LIN {X 0,Y 453.11,Z 853.7,A -85,B 0,C 180,E1 14752.247,E2 14752.247} C_VEL
LIN {X 0,Y 449.682,Z 846.893,A -85,B 0,C 180,E1 14758.978,E2 14758.978} C_VEL
LIN {X 0,Y 456.132,Z 857.359,A -85,B 0,C 180,E1 14770.845,E2 14770.845} C_VEL
LIN {X 0,Y 467.562,Z 871.986,A -85,B 0,C 180,E1 14777.472,E2 14777.472} C_VEL
LIN {X 0,Y 488.075,Z 901.104,A -85,B 0,C 180,E1 14785.371,E2 14785.371} C_VEL
LIN {X 0,Y 511.745,Z 944.514,A -85,B 0,C 180,E1 14792.88,E2 14792.88} C_VEL
LIN {X 0,Y 522.504,Z 975.983,A -85,B 0,C 180,E1 14796.793,E2 14796.793} C_VEL
LIN {X 0,Y 504.777,Z 1049.312,A -85,B 0,C 180,E1 14800.922,E2 14800.922} C_VEL
LIN {X 0,Y 484.838,Z 1113.765,A -85,B 0,C 180,E1 14806.768,E2 14806.768} C_VEL
LIN {X 0,Y 466.012,Z 1168.211,A -85,B 0,C 180,E1 14814.348,E2 14814.348} C_VEL
LIN {X 0,Y 452.106,Z 1211.205,A -85,B 0,C 180,E1 14823.581,E2 14823.581} C_VEL
LIN {X 0,Y 445.258,Z 1240.185,A -85,B 0,C 180,E1 14833.662,E2 14833.662} C_VEL
LIN {X 0,Y 443.189,Z 1254.354,A -85,B 0,C 180,E1 14843.114,E2 14843.114} C_VEL
LIN {X 0,Y 443.168,Z 1257.3,A -85,B 0,C 180,E1 14850.981,E2 14850.981} C_VEL
LIN {X 0,Y 443.526,Z 1251.078,A -85,B 0,C 180,E1 14859.854,E2 14859.854} C_VEL
LIN {X 0,Y 446.199,Z 1232.875,A -85,B 0,C 180,E1 14869.373,E2 14869.373} C_VEL
LIN {X 0,Y 455.013,Z 1201.001,A -85,B 0,C 180,E1 14878.932,E2 14878.932} C_VEL
LIN {X 0,Y 470.637,Z 1154.491,A -85,B 0,C 180,E1 14887.802,E2 14887.802} C_VEL
LIN {X 0,Y 490.557,Z 1096.151,A -85,B 0,C 180,E1 14895.007,E2 14895.007} C_VEL
LIN {X 0,Y 510.312,Z 1029.556,A -85,B 0,C 180,E1 14900.284,E2 14900.284} C_VEL
LIN {X 0,Y 522.312,Z 970.799,A -85,B 0,C 180,E1 14903.513,E2 14903.513} C_VEL
LIN {X 0,Y 500.816,Z 922.884,A -85,B 0,C 180,E1 14910.405,E2 14910.405} C_VEL
LIN {X 0,Y 478.038,Z 886.237,A -85,B 0,C 180,E1 14918.038,E2 14918.038} C_VEL
LIN {X 0,Y 460.008,Z 861.655,A -85,B 0,C 180,E1 14926.343,E2 14926.343} C_VEL
LIN {X 0,Y 453.526,Z 853.849,A -85,B 0,C 180,E1 14931.155,E2 14931.155} C_VEL
LIN {X 0,Y 449.33,Z 846.815,A -85,B 0,C 180,E1 14939.088,E2 14939.088} C_VEL
LIN {X 0,Y 455.483,Z 855.768,A -85,B 0,C 180,E1 14950.006,E2 14950.006} C_VEL
LIN {X 0,Y 468.677,Z 873.827,A -85,B 0,C 180,E1 14957.65,E2 14957.65} C_VEL
LIN {X 0,Y 490.163,Z 903.109,A -85,B 0,C 180,E1 14965.368,E2 14965.368} C_VEL
LIN {X 0,Y 516.111,Z 949.406,A -85,B 0,C 180,E1 14972.898,E2 14972.898} C_VEL
LIN {X 0,Y 525.972,Z 974.905,A -85,B 0,C 180,E1 14975.93,E2 14975.93} C_VEL
LIN {X 0,Y 510.004,Z 1047.435,A -85,B 0,C 180,E1 14979.293,E2 14979.293} C_VEL
LIN {X 0,Y 490.013,Z 1116.733,A -85,B 0,C 180,E1 14984.599,E2 14984.599} C_VEL
LIN {X 0,Y 470.658,Z 1176.48,A -85,B 0,C 180,E1 14991.727,E2 14991.727} C_VEL
LIN {X 0,Y 455.499,Z 1224.574,A -85,B 0,C 180,E1 15000.429,E2 15000.429} C_VEL
LIN {X 0,Y 446.704,Z 1259.254,A -85,B 0,C 180,E1 15010.133,E2 15010.133} C_VEL
LIN {X 0,Y 443.508,Z 1278.435,A -85,B 0,C 180,E1 15019.149,E2 15019.149} C_VEL
LIN {X 0,Y 443.111,Z 1285.921,A -85,B 0,C 180,E1 15027.055,E2 15027.055} C_VEL
LIN {X 0,Y 443.189,Z 1284.856,A -85,B 0,C 180,E1 15034.913,E2 15034.913} C_VEL
LIN {X 0,Y 443.981,Z 1273.992,A -85,B 0,C 180,E1 15043.49,E2 15043.49} C_VEL
LIN {X 0,Y 437.709,Z 1265,A -85,B 0,C 180,E1 15047.886,E2 15047.886} C_VEL
LIN {X 0,Y 445.554,Z 1232.734,A -85,B 0,C 180,E1 15058.106,E2 15058.106} C_VEL
LIN {X 0,Y 460.411,Z 1186.788,A -85,B 0,C 180,E1 15067.293,E2 15067.293} C_VEL
LIN {X 0,Y 480.299,Z 1128.807,A -85,B 0,C 180,E1 15074.859,E2 15074.859} C_VEL
LIN {X 0,Y 501.097,Z 1060.927,A -85,B 0,C 180,E1 15080.584,E2 15080.584} C_VEL
LIN {X 0,Y 519.127,Z 985.374,A -85,B 0,C 180,E1 15084.445,E2 15084.445} C_VEL
LIN {X 0,Y 519.955,Z 974.55,A -85,B 0,C 180,E1 15085.007,E2 15085.007} C_VEL
LIN {X 0,Y 497.411,Z 926.333,A -85,B 0,C 180,E1 15091.89,E2 15091.89} C_VEL
LIN {X 0,Y 474.399,Z 890.834,A -85,B 0,C 180,E1 15099.591,E2 15099.591} C_VEL
LIN {X 0,Y 457.866,Z 869.113,A -85,B 0,C 180,E1 15107.615,E2 15107.615} C_VEL
LIN {X 0,Y 451.9,Z 861.515,A -85,B 0,C 180,E1 15112.469,E2 15112.469} C_VEL
LIN {X 0,Y 448.631,Z 854.888,A -85,B 0,C 180,E1 15120.913,E2 15120.913} C_VEL
LIN {X 0,Y 455.13,Z 865.662,A -85,B 0,C 180,E1 15130.869,E2 15130.869} C_VEL
LIN {X 0,Y 466.056,Z 880.022,A -85,B 0,C 180,E1 15137.347,E2 15137.347} C_VEL
LIN {X 0,Y 486.826,Z 910.227,A -85,B 0,C 180,E1 15145.543,E2 15145.543} C_VEL
LIN {X 0,Y 508.661,Z 953.325,A -85,B 0,C 180,E1 15152.921,E2 15152.921} C_VEL
LIN {X 0,Y 517.223,Z 978.635,A -85,B 0,C 180,E1 15156.18,E2 15156.18} C_VEL
LIN {X 0,Y 499.121,Z 1050.75,A -85,B 0,C 180,E1 15160.297,E2 15160.297} C_VEL
LIN {X 0,Y 478.45,Z 1115.183,A -85,B 0,C 180,E1 15166.219,E2 15166.219} C_VEL
LIN {X 0,Y 459.135,Z 1168.858,A -85,B 0,C 180,E1 15173.807,E2 15173.807} C_VEL
LIN {X 0,Y 444.616,Z 1211.478,A -85,B 0,C 180,E1 15183.101,E2 15183.101} C_VEL
LIN {X 0,Y 437.447,Z 1240.451,A -85,B 0,C 180,E1 15193.362,E2 15193.362} C_VEL
LIN {X 0,Y 435.219,Z 1254.617,A -85,B 0,C 180,E1 15202.987,E2 15202.987} C_VEL
LIN {X 0,Y 435.171,Z 1257.563,A -85,B 0,C 180,E1 15210.999,E2 15210.999} C_VEL
LIN {X 0,Y 435.567,Z 1251.344,A -85,B 0,C 180,E1 15220.036,E2 15220.036} C_VEL
LIN {X 0,Y 438.475,Z 1233.146,A -85,B 0,C 180,E1 15229.728,E2 15229.728} C_VEL
LIN {X 0,Y 447.767,Z 1201.276,A -85,B 0,C 180,E1 15239.446,E2 15239.446} C_VEL
LIN {X 0,Y 464.103,Z 1154.767,A -85,B 0,C 180,E1 15248.431,E2 15248.431} C_VEL
LIN {X 0,Y 484.889,Z 1096.018,A -85,B 0,C 180,E1 15255.738,E2 15255.738} C_VEL
LIN {X 0,Y 504.973,Z 1030.479,A -85,B 0,C 180,E1 15260.953,E2 15260.953} C_VEL
LIN {X 0,Y 516.768,Z 974.458,A -85,B 0,C 180,E1 15264.101,E2 15264.101} C_VEL
LIN {X 0,Y 496.134,Z 927.061,A -85,B 0,C 180,E1 15271.146,E2 15271.146} C_VEL
LIN {X 0,Y 473.874,Z 890.484,A -85,B 0,C 180,E1 15279.129,E2 15279.129} C_VEL
LIN {X 0,Y 457.673,Z 868.684,A -85,B 0,C 180,E1 15287.126,E2 15287.126} C_VEL
LIN {X 0,Y 452.049,Z 861.472,A -85,B 0,C 180,E1 15291.612,E2 15291.612} C_VEL
LIN {X 0,Y 448.355,Z 854.755,A -85,B 0,C 180,E1 15299.086,E2 15299.086} C_VEL
LIN {X 0,Y 454.259,Z 863.811,A -85,B 0,C 180,E1 15309.851,E2 15309.851} C_VEL
LIN {X 0,Y 467.341,Z 881.776,A -85,B 0,C 180,E1 15317.531,E2 15317.531} C_VEL
LIN {X 0,Y 488.148,Z 911.534,A -85,B 0,C 180,E1 15325.295,E2 15325.295} C_VEL
LIN {X 0,Y 512.404,Z 956.503,A -85,B 0,C 180,E1 15332.685,E2 15332.685} C_VEL
LIN {X 0,Y 520.374,Z 979.416,A -85,B 0,C 180,E1 15335.378,E2 15335.378} C_VEL
LIN {X 0,Y 503.728,Z 1051.271,A -85,B 0,C 180,E1 15338.825,E2 15338.825} C_VEL
LIN {X 0,Y 482.851,Z 1120.512,A -85,B 0,C 180,E1 15344.293,E2 15344.293} C_VEL
LIN {X 0,Y 463.009,Z 1179.262,A -85,B 0,C 180,E1 15351.541,E2 15351.541} C_VEL
LIN {X 0,Y 447.361,Z 1227.03,A -85,B 0,C 180,E1 15360.525,E2 15360.525} C_VEL
LIN {X 0,Y 438.59,Z 1260.356,A -85,B 0,C 180,E1 15370.277,E2 15370.277} C_VEL
LIN {X 0,Y 435.425,Z 1279.547,A -85,B 0,C 180,E1 15379.961,E2 15379.961} C_VEL
LIN {X 0,Y 435.469,Z 1286.143,A -85,B 0,C 180,E1 15389.002,E2 15389.002} C_VEL
LIN {X 0,Y 435.223,Z 1282.035,A -85,B 0,C 180,E1 15398.021,E2 15398.021} C_VEL
LIN {X 0,Y 437.709,Z 1265,A -85,B 0,C 180,E1 15407.886,E2 15407.886} C_VEL
LIN {X 0,Y 431.738,Z 1254.138,A -85,B 0,C 180,E1 15412.282,E2 15412.282} C_VEL
LIN {X 0,Y 442.101,Z 1219.334,A -85,B 0,C 180,E1 15421.759,E2 15421.759} C_VEL
LIN {X 0,Y 459.976,Z 1168.875,A -85,B 0,C 180,E1 15430.636,E2 15430.636} C_VEL
LIN {X 0,Y 481.519,Z 1107.411,A -85,B 0,C 180,E1 15437.644,E2 15437.644} C_VEL
LIN {X 0,Y 501.982,Z 1039.364,A -85,B 0,C 180,E1 15442.593,E2 15442.593} C_VEL
LIN {X 0,Y 514.55,Z 978.138,A -85,B 0,C 180,E1 15445.62,E2 15445.62} C_VEL
LIN {X 0,Y 493.082,Z 931.355,A -85,B 0,C 180,E1 15452.528,E2 15452.528} C_VEL
LIN {X 0,Y 471.954,Z 897.803,A -85,B 0,C 180,E1 15460.033,E2 15460.033} C_VEL
LIN {X 0,Y 456.328,Z 876.653,A -85,B 0,C 180,E1 15467.951,E2 15467.951} C_VEL
LIN {X 0,Y 450.479,Z 869.111,A -85,B 0,C 180,E1 15472.932,E2 15472.932} C_VEL
LIN {X 0,Y 447.656,Z 862.828,A -85,B 0,C 180,E1 15480.915,E2 15480.915} C_VEL
LIN {X 0,Y 453.995,Z 873.676,A -85,B 0,C 180,E1 15490.779,E2 15490.779} C_VEL
LIN {X 0,Y 464.875,Z 888.499,A -85,B 0,C 180,E1 15497.392,E2 15497.392} C_VEL
LIN {X 0,Y 484.206,Z 918.023,A -85,B 0,C 180,E1 15505.394,E2 15505.394} C_VEL
LIN {X 0,Y 504.697,Z 960.166,A -85,B 0,C 180,E1 15512.7,E2 15512.7} C_VEL
LIN {X 0,Y 511.792,Z 982.53,A -85,B 0,C 180,E1 15515.615,E2 15515.615} C_VEL
LIN {X 0,Y 492.699,Z 1054.947,A -85,B 0,C 180,E1 15519.854,E2 15519.854} C_VEL
LIN {X 0,Y 471.361,Z 1118.752,A -85,B 0,C 180,E1 15525.899,E2 15525.899} C_VEL
LIN {X 0,Y 450.971,Z 1173.22,A -85,B 0,C 180,E1 15533.906,E2 15533.906} C_VEL
LIN {X 0,Y 436.26,Z 1215.391,A -85,B 0,C 180,E1 15543.66,E2 15543.66} C_VEL
LIN {X 0,Y 429.385,Z 1241.838,A -85,B 0,C 180,E1 15553.569,E2 15553.569} C_VEL
LIN {X 0,Y 427.232,Z 1254.881,A -85,B 0,C 180,E1 15562.855,E2 15562.855} C_VEL
LIN {X 0,Y 427.202,Z 1257.824,A -85,B 0,C 180,E1 15571.017,E2 15571.017} C_VEL
LIN {X 0,Y 427.586,Z 1251.611,A -85,B 0,C 180,E1 15580.225,E2 15580.225} C_VEL
LIN {X 0,Y 430.757,Z 1233.435,A -85,B 0,C 180,E1 15590.089,E2 15590.089} C_VEL
LIN {X 0,Y 440.547,Z 1201.552,A -85,B 0,C 180,E1 15599.977,E2 15599.977} C_VEL
LIN {X 0,Y 457.389,Z 1155.709,A -85,B 0,C 180,E1 15608.972,E2 15608.972} C_VEL
LIN {X 0,Y 478.774,Z 1097.425,A -85,B 0,C 180,E1 15616.331,E2 15616.331} C_VEL
LIN {X 0,Y 499.892,Z 1030.798,A -85,B 0,C 180,E1 15621.672,E2 15621.672} C_VEL
LIN {X 0,Y 511.857,Z 979.714,A -85,B 0,C 180,E1 15624.486,E2 15624.486} C_VEL
LIN {X 0,Y 492.306,Z 932.966,A -85,B 0,C 180,E1 15631.591,E2 15631.591} C_VEL
LIN {X 0,Y 471.233,Z 897.38,A -85,B 0,C 180,E1 15639.561,E2 15639.561} C_VEL
LIN {X 0,Y 455.949,Z 876.053,A -85,B 0,C 180,E1 15647.565,E2 15647.565} C_VEL
LIN {X 0,Y 450.835,Z 869.282,A -85,B 0,C 180,E1 15651.833,E2 15651.833} C_VEL
LIN {X 0,Y 447.381,Z 862.695,A -85,B 0,C 180,E1 15659.084,E2 15659.084} C_VEL
LIN {X 0,Y 453.357,Z 872.65,A -85,B 0,C 180,E1 15669.992,E2 15669.992} C_VEL
LIN {X 0,Y 465.347,Z 889.013,A -85,B 0,C 180,E1 15677.181,E2 15677.181} C_VEL
LIN {X 0,Y 485.623,Z 918.952,A -85,B 0,C 180,E1 15685.063,E2 15685.063} C_VEL
LIN {X 0,Y 508.669,Z 963.487,A -85,B 0,C 180,E1 15692.456,E2 15692.456} C_VEL
LIN {X 0,Y 514.971,Z 982.994,A -85,B 0,C 180,E1 15694.776,E2 15694.776} C_VEL
LIN {X 0,Y 497.853,Z 1053.719,A -85,B 0,C 180,E1 15698.257,E2 15698.257} C_VEL
LIN {X 0,Y 476.308,Z 1122.453,A -85,B 0,C 180,E1 15703.794,E2 15703.794} C_VEL
LIN {X 0,Y 456.004,Z 1180.218,A -85,B 0,C 180,E1 15711.071,E2 15711.071} C_VEL
LIN {X 0,Y 439.71,Z 1227.863,A -85,B 0,C 180,E1 15720.245,E2 15720.245} C_VEL
LIN {X 0,Y 430.453,Z 1261.457,A -85,B 0,C 180,E1 15730.425,E2 15730.425} C_VEL
LIN {X 0,Y 427.443,Z 1279.281,A -85,B 0,C 180,E1 15739.772,E2 15739.772} C_VEL
LIN {X 0,Y 427.486,Z 1285.881,A -85,B 0,C 180,E1 15748.983,E2 15748.983} C_VEL
LIN {X 0,Y 427.261,Z 1281.771,A -85,B 0,C 180,E1 15758.171,E2 15758.171} C_VEL
LIN {X 0,Y 430.028,Z 1264.044,A -85,B 0,C 180,E1 15768.526,E2 15768.526} C_VEL
LIN {X 0,Y 431.738,Z 1254.138,A -85,B 0,C 180,E1 15772.282,E2 15772.282} C_VEL
LIN {X 0,Y 428.136,Z 1241.283,A -85,B 0,C 180,E1 15776.671,E2 15776.671} C_VEL
LIN {X 0,Y 442.508,Z 1198.865,A -85,B 0,C 180,E1 15786.394,E2 15786.394} C_VEL
LIN {X 0,Y 463.058,Z 1143.42,A -85,B 0,C 180,E1 15794.606,E2 15794.606} C_VEL
LIN {X 0,Y 485.732,Z 1077.138,A -85,B 0,C 180,E1 15800.89,E2 15800.89} C_VEL
LIN {X 0,Y 505.9,Z 1003.625,A -85,B 0,C 180,E1 15805.141,E2 15805.141} C_VEL
LIN {X 0,Y 509.324,Z 982.117,A -85,B 0,C 180,E1 15806.2,E2 15806.2} C_VEL
LIN {X 0,Y 488.656,Z 936.006,A -85,B 0,C 180,E1 15813.237,E2 15813.237} C_VEL
LIN {X 0,Y 468.949,Z 904.053,A -85,B 0,C 180,E1 15820.699,E2 15820.699} C_VEL
LIN {X 0,Y 454.583,Z 884.034,A -85,B 0,C 180,E1 15828.392,E2 15828.392} C_VEL
LIN {X 0,Y 449.084,Z 876.743,A -85,B 0,C 180,E1 15833.397,E2 15833.397} C_VEL
LIN {X 0,Y 446.683,Z 870.754,A -85,B 0,C 180,E1 15840.917,E2 15840.917} C_VEL
LIN {X 0,Y 452.859,Z 881.852,A -85,B 0,C 180,E1 15850.806,E2 15850.806} C_VEL
LIN {X 0,Y 465.789,Z 899.557,A -85,B 0,C 180,E1 15858.522,E2 15858.522} C_VEL
LIN {X 0,Y 485.836,Z 933.76,A -85,B 0,C 180,E1 15866.867,E2 15866.867} C_VEL
LIN {X 0,Y 504.507,Z 977.636,A -85,B 0,C 180,E1 15874.019,E2 15874.019} C_VEL
LIN {X 0,Y 505.912,Z 988.262,A -85,B 0,C 180,E1 15875.126,E2 15875.126} C_VEL
LIN {X 0,Y 485.863,Z 1060.395,A -85,B 0,C 180,E1 15879.521,E2 15879.521} C_VEL
LIN {X 0,Y 463.572,Z 1123.832,A -85,B 0,C 180,E1 15885.777,E2 15885.777} C_VEL
LIN {X 0,Y 443.176,Z 1176.189,A -85,B 0,C 180,E1 15893.798,E2 15893.798} C_VEL
LIN {X 0,Y 428.288,Z 1217.361,A -85,B 0,C 180,E1 15903.699,E2 15903.699} C_VEL
LIN {X 0,Y 420.937,Z 1244.017,A -85,B 0,C 180,E1 15914.306,E2 15914.306} C_VEL
LIN {X 0,Y 419.162,Z 1256.093,A -85,B 0,C 180,E1 15923.903,E2 15923.903} C_VEL
LIN {X 0,Y 419.202,Z 1257.635,A -85,B 0,C 180,E1 15933.113,E2 15933.113} C_VEL
LIN {X 0,Y 419.846,Z 1249.304,A -85,B 0,C 180,E1 15942.354,E2 15942.354} C_VEL
LIN {X 0,Y 424.922,Z 1228.23,A -85,B 0,C 180,E1 15952.585,E2 15952.585} C_VEL
LIN {X 0,Y 436.897,Z 1193.077,A -85,B 0,C 180,E1 15962.587,E2 15962.587} C_VEL
LIN {X 0,Y 455.094,Z 1145.757,A -85,B 0,C 180,E1 15971.193,E2 15971.193} C_VEL
LIN {X 0,Y 477.176,Z 1086.488,A -85,B 0,C 180,E1 15978.141,E2 15978.141} C_VEL
LIN {X 0,Y 498.343,Z 1018.96,A -85,B 0,C 180,E1 15983.144,E2 15983.144} C_VEL
LIN {X 0,Y 506.159,Z 982.556,A -85,B 0,C 180,E1 15985.203,E2 15985.203} C_VEL
LIN {X 0,Y 487.494,Z 937.272,A -85,B 0,C 180,E1 15992.359,E2 15992.359} C_VEL
LIN {X 0,Y 468.289,Z 903.91,A -85,B 0,C 180,E1 16000.107,E2 16000.107} C_VEL
LIN {X 0,Y 454.043,Z 883.251,A -85,B 0,C 180,E1 16008.063,E2 16008.063} C_VEL
LIN {X 0,Y 449.166,Z 876.737,A -85,B 0,C 180,E1 16012.535,E2 16012.535} C_VEL
LIN {X 0,Y 446.406,Z 870.635,A -85,B 0,C 180,E1 16019.082,E2 16019.082} C_VEL
LIN {X 0,Y 452.407,Z 881.126,A -85,B 0,C 180,E1 16030.075,E2 16030.075} C_VEL
LIN {X 0,Y 464.066,Z 897.184,A -85,B 0,C 180,E1 16037.168,E2 16037.168} C_VEL
LIN {X 0,Y 483.946,Z 927.901,A -85,B 0,C 180,E1 16045.164,E2 16045.164} C_VEL
LIN {X 0,Y 504.916,Z 970.827,A -85,B 0,C 180,E1 16052.291,E2 16052.291} C_VEL
LIN {X 0,Y 509.389,Z 987.554,A -85,B 0,C 180,E1 16054.207,E2 16054.207} C_VEL
LIN {X 0,Y 491.278,Z 1059.063,A -85,B 0,C 180,E1 16057.866,E2 16057.866} C_VEL
LIN {X 0,Y 469.06,Z 1126.651,A -85,B 0,C 180,E1 16063.514,E2 16063.514} C_VEL
LIN {X 0,Y 447.703,Z 1184.738,A -85,B 0,C 180,E1 16071.148,E2 16071.148} C_VEL
LIN {X 0,Y 431.377,Z 1230.805,A -85,B 0,C 180,E1 16080.483,E2 16080.483} C_VEL
LIN {X 0,Y 421.966,Z 1263.766,A -85,B 0,C 180,E1 16091.108,E2 16091.108} C_VEL
LIN {X 0,Y 419.361,Z 1280.267,A -85,B 0,C 180,E1 16100.625,E2 16100.625} C_VEL
LIN {X 0,Y 419.478,Z 1285.618,A -85,B 0,C 180,E1 16108.964,E2 16108.964} C_VEL
LIN {X 0,Y 419.289,Z 1281.506,A -85,B 0,C 180,E1 16118.328,E2 16118.328} C_VEL
LIN {X 0,Y 422.198,Z 1263.772,A -85,B 0,C 180,E1 16128.882,E2 16128.882} C_VEL
LIN {X 0,Y 428.136,Z 1241.283,A -85,B 0,C 180,E1 16136.671,E2 16136.671} C_VEL
LIN {X 0,Y 424.983,Z 1226.871,A -85,B 0,C 180,E1 16141.011,E2 16141.011} C_VEL
LIN {X 0,Y 442.772,Z 1179.823,A -85,B 0,C 180,E1 16150.298,E2 16150.298} C_VEL
LIN {X 0,Y 465.383,Z 1120.782,A -85,B 0,C 180,E1 16157.803,E2 16157.803} C_VEL
LIN {X 0,Y 487.983,Z 1052.959,A -85,B 0,C 180,E1 16163.273,E2 16163.273} C_VEL
LIN {X 0,Y 504.383,Z 986.954,A -85,B 0,C 180,E1 16166.678,E2 16166.678} C_VEL
LIN {X 0,Y 484.758,Z 941.385,A -85,B 0,C 180,E1 16173.806,E2 16173.806} C_VEL
LIN {X 0,Y 465.57,Z 909.733,A -85,B 0,C 180,E1 16181.479,E2 16181.479} C_VEL
LIN {X 0,Y 451.998,Z 890.364,A -85,B 0,C 180,E1 16189.427,E2 16189.427} C_VEL
LIN {X 0,Y 447.433,Z 884.16,A -85,B 0,C 180,E1 16194.105,E2 16194.105} C_VEL
LIN {X 0,Y 445.678,Z 878.763,A -85,B 0,C 180,E1 16200.919,E2 16200.919} C_VEL
LIN {X 0,Y 451.481,Z 889.666,A -85,B 0,C 180,E1 16210.656,E2 16210.656} C_VEL
LIN {X 0,Y 464.082,Z 908.098,A -85,B 0,C 180,E1 16218.531,E2 16218.531} C_VEL
LIN {X 0,Y 482.695,Z 941.071,A -85,B 0,C 180,E1 16226.677,E2 16226.677} C_VEL
LIN {X 0,Y 500.722,Z 985.928,A -85,B 0,C 180,E1 16234.034,E2 16234.034} C_VEL
LIN {X 0,Y 482.132,Z 1056.434,A -85,B 0,C 180,E1 16238.44,E2 16238.44} C_VEL
LIN {X 0,Y 458.972,Z 1121.016,A -85,B 0,C 180,E1 16244.671,E2 16244.671} C_VEL
LIN {X 0,Y 437.153,Z 1174.802,A -85,B 0,C 180,E1 16252.823,E2 16252.823} C_VEL
LIN {X 0,Y 421.163,Z 1216.307,A -85,B 0,C 180,E1 16262.765,E2 16262.765} C_VEL
LIN {X 0,Y 413.68,Z 1242.49,A -85,B 0,C 180,E1 16272.986,E2 16272.986} C_VEL
LIN {X 0,Y 411.291,Z 1255.407,A -85,B 0,C 180,E1 16282.577,E2 16282.577} C_VEL
LIN {X 0,Y 411.22,Z 1258.349,A -85,B 0,C 180,E1 16291.057,E2 16291.057} C_VEL
LIN {X 0,Y 411.654,Z 1252.145,A -85,B 0,C 180,E1 16300.625,E2 16300.625} C_VEL
LIN {X 0,Y 415.575,Z 1233.49,A -85,B 0,C 180,E1 16311.065,E2 16311.065} C_VEL
LIN {X 0,Y 426.91,Z 1200.435,A -85,B 0,C 180,E1 16321.504,E2 16321.504} C_VEL
LIN {X 0,Y 445.617,Z 1153.895,A -85,B 0,C 180,E1 16330.688,E2 16330.688} C_VEL
LIN {X 0,Y 468.355,Z 1095.897,A -85,B 0,C 180,E1 16337.998,E2 16337.998} C_VEL
LIN {X 0,Y 490.295,Z 1030.191,A -85,B 0,C 180,E1 16343.24,E2 16343.24} C_VEL
LIN {X 0,Y 500.914,Z 986.653,A -85,B 0,C 180,E1 16345.763,E2 16345.763} C_VEL
LIN {X 0,Y 482.941,Z 941.789,A -85,B 0,C 180,E1 16353.086,E2 16353.086} C_VEL
LIN {X 0,Y 464.65,Z 909.17,A -85,B 0,C 180,E1 16361.02,E2 16361.02} C_VEL
LIN {X 0,Y 450.279,Z 886.019,A -85,B 0,C 180,E1 16370.357,E2 16370.357} C_VEL
LIN {X 0,Y 445.416,Z 878.564,A -85,B 0,C 180,E1 16379.08,E2 16379.08} C_VEL
LIN {X 0,Y 451.162,Z 889.201,A -85,B 0,C 180,E1 16390.042,E2 16390.042} C_VEL
LIN {X 0,Y 464.107,Z 906.937,A -85,B 0,C 180,E1 16397.842,E2 16397.842} C_VEL
LIN {X 0,Y 484.623,Z 941.699,A -85,B 0,C 180,E1 16406.214,E2 16406.214} C_VEL
LIN {X 0,Y 504.277,Z 986.818,A -85,B 0,C 180,E1 16413.309,E2 16413.309} C_VEL
LIN {X 0,Y 485.4,Z 1061.581,A -85,B 0,C 180,E1 16417.29,E2 16417.29} C_VEL
LIN {X 0,Y 462.363,Z 1128.919,A -85,B 0,C 180,E1 16423.044,E2 16423.044} C_VEL
LIN {X 0,Y 440.375,Z 1186.417,A -85,B 0,C 180,E1 16430.797,E2 16430.797} C_VEL
LIN {X 0,Y 423.342,Z 1232.525,A -85,B 0,C 180,E1 16440.458,E2 16440.458} C_VEL
LIN {X 0,Y 413.84,Z 1264.676,A -85,B 0,C 180,E1 16451.278,E2 16451.278} C_VEL
LIN {X 0,Y 411.369,Z 1281.243,A -85,B 0,C 180,E1 16461.512,E2 16461.512} C_VEL
LIN {X 0,Y 411.103,Z 1285.343,A -85,B 0,C 180,E1 16471.059,E2 16471.059} C_VEL
LIN {X 0,Y 411.654,Z 1278.753,A -85,B 0,C 180,E1 16480.626,E2 16480.626} C_VEL
LIN {X 0,Y 415.092,Z 1259.071,A -85,B 0,C 180,E1 16491.078,E2 16491.078} C_VEL
LIN {X 0,Y 424.983,Z 1226.871,A -85,B 0,C 180,E1 16501.011,E2 16501.011} C_VEL
LIN {X 0,Y 421.507,Z 1216.859,A -85,B 0,C 180,E1 16503.926,E2 16503.926} C_VEL
LIN {X 0,Y 441.949,Z 1166.018,A -85,B 0,C 180,E1 16513.057,E2 16513.057} C_VEL
LIN {X 0,Y 465.485,Z 1105.339,A -85,B 0,C 180,E1 16520.035,E2 16520.035} C_VEL
LIN {X 0,Y 487.421,Z 1038.62,A -85,B 0,C 180,E1 16524.887,E2 16524.887} C_VEL
LIN {X 0,Y 498.962,Z 990.551,A -85,B 0,C 180,E1 16527.318,E2 16527.318} C_VEL
LIN {X 0,Y 480.676,Z 946.759,A -85,B 0,C 180,E1 16534.409,E2 16534.409} C_VEL
LIN {X 0,Y 461.545,Z 913.861,A -85,B 0,C 180,E1 16542.673,E2 16542.673} C_VEL
LIN {X 0,Y 448.223,Z 893.562,A -85,B 0,C 180,E1 16551.917,E2 16551.917} C_VEL
LIN {X 0,Y 444.498,Z 886.853,A -85,B 0,C 180,E1 16560.922,E2 16560.922} C_VEL
LIN {X 0,Y 450.058,Z 897.606,A -85,B 0,C 180,E1 16570.567,E2 16570.567} C_VEL
LIN {X 0,Y 462.111,Z 916.161,A -85,B 0,C 180,E1 16578.463,E2 16578.463} C_VEL
LIN {X 0,Y 479.554,Z 948.493,A -85,B 0,C 180,E1 16586.492,E2 16586.492} C_VEL
LIN {X 0,Y 495.847,Z 991.539,A -85,B 0,C 180,E1 16593.693,E2 16593.693} C_VEL
LIN {X 0,Y 474.592,Z 1063.824,A -85,B 0,C 180,E1 16598.232,E2 16598.232} C_VEL
LIN {X 0,Y 450.817,Z 1126.838,A -85,B 0,C 180,E1 16604.626,E2 16604.626} C_VEL
LIN {X 0,Y 429.012,Z 1178.689,A -85,B 0,C 180,E1 16612.88,E2 16612.88} C_VEL
LIN {X 0,Y 412.915,Z 1219.374,A -85,B 0,C 180,E1 16623.151,E2 16623.151} C_VEL
LIN {X 0,Y 405.277,Z 1244.549,A -85,B 0,C 180,E1 16633.683,E2 16633.683} C_VEL
LIN {X 0,Y 403.328,Z 1255.67,A -85,B 0,C 180,E1 16642.429,E2 16642.429} C_VEL
LIN {X 0,Y 403.221,Z 1258.612,A -85,B 0,C 180,E1 16651.078,E2 16651.078} C_VEL
LIN {X 0,Y 403.695,Z 1252.411,A -85,B 0,C 180,E1 16660.837,E2 16660.837} C_VEL
LIN {X 0,Y 407.945,Z 1233.761,A -85,B 0,C 180,E1 16671.478,E2 16671.478} C_VEL
LIN {X 0,Y 420.179,Z 1200.031,A -85,B 0,C 180,E1 16682.263,E2 16682.263} C_VEL
LIN {X 0,Y 439.979,Z 1152.74,A -85,B 0,C 180,E1 16691.621,E2 16691.621} C_VEL
LIN {X 0,Y 463.099,Z 1095.637,A -85,B 0,C 180,E1 16698.808,E2 16698.808} C_VEL
LIN {X 0,Y 486.044,Z 1028.754,A -85,B 0,C 180,E1 16704.108,E2 16704.108} C_VEL
LIN {X 0,Y 495.55,Z 990.756,A -85,B 0,C 180,E1 16706.327,E2 16706.327} C_VEL
LIN {X 0,Y 478.862,Z 947.112,A -85,B 0,C 180,E1 16713.663,E2 16713.663} C_VEL
LIN {X 0,Y 460.882,Z 913.691,A -85,B 0,C 180,E1 16722.093,E2 16722.093} C_VEL
LIN {X 0,Y 448.301,Z 893.576,A -85,B 0,C 180,E1 16731.051,E2 16731.051} C_VEL
LIN {X 0,Y 444.261,Z 886.48,A -85,B 0,C 180,E1 16739.078,E2 16739.078} C_VEL
LIN {X 0,Y 449.852,Z 897.141,A -85,B 0,C 180,E1 16749.948,E2 16749.948} C_VEL
LIN {X 0,Y 462.403,Z 915.428,A -85,B 0,C 180,E1 16757.848,E2 16757.848} C_VEL
LIN {X 0,Y 481.415,Z 948.741,A -85,B 0,C 180,E1 16765.956,E2 16765.956} C_VEL
LIN {X 0,Y 499.165,Z 991.371,A -85,B 0,C 180,E1 16772.801,E2 16772.801} C_VEL
LIN {X 0,Y 479.437,Z 1064.377,A -85,B 0,C 180,E1 16776.72,E2 16776.72} C_VEL
LIN {X 0,Y 455.846,Z 1130.782,A -85,B 0,C 180,E1 16782.515,E2 16782.515} C_VEL
LIN {X 0,Y 433.05,Z 1188.092,A -85,B 0,C 180,E1 16790.431,E2 16790.431} C_VEL
LIN {X 0,Y 415.887,Z 1232.683,A -85,B 0,C 180,E1 16800.005,E2 16800.005} C_VEL
LIN {X 0,Y 406.087,Z 1264.407,A -85,B 0,C 180,E1 16810.907,E2 16810.907} C_VEL
LIN {X 0,Y 403.377,Z 1280.978,A -85,B 0,C 180,E1 16821.342,E2 16821.342} C_VEL
LIN {X 0,Y 403.102,Z 1285.08,A -85,B 0,C 180,E1 16831.08,E2 16831.08} C_VEL
LIN {X 0,Y 403.675,Z 1278.487,A -85,B 0,C 180,E1 16840.839,E2 16840.839} C_VEL
LIN {X 0,Y 407.299,Z 1258.797,A -85,B 0,C 180,E1 16851.501,E2 16851.501} C_VEL
LIN {X 0,Y 418.027,Z 1225.906,A -85,B 0,C 180,E1 16861.776,E2 16861.776} C_VEL
LIN {X 0,Y 421.507,Z 1216.859,A -85,B 0,C 180,E1 16863.926,E2 16863.926} C_VEL
LIN {X 0,Y 421.759,Z 1199.506,A -85,B 0,C 180,E1 16868.144,E2 16868.144} C_VEL
LIN {X 0,Y 444.381,Z 1145.239,A -85,B 0,C 180,E1 16876.549,E2 16876.549} C_VEL
LIN {X 0,Y 468.851,Z 1080.733,A -85,B 0,C 180,E1 16882.899,E2 16882.899} C_VEL
LIN {X 0,Y 491.004,Z 1008.017,A -85,B 0,C 180,E1 16887.24,E2 16887.24} C_VEL
LIN {X 0,Y 493.422,Z 993.646,A -85,B 0,C 180,E1 16888.047,E2 16888.047} C_VEL
LIN {X 0,Y 476.029,Z 950.992,A -85,B 0,C 180,E1 16895.229,E2 16895.229} C_VEL
LIN {X 0,Y 458.477,Z 920.25,A -85,B 0,C 180,E1 16903.384,E2 16903.384} C_VEL
LIN {X 0,Y 446.758,Z 901.345,A -85,B 0,C 180,E1 16912.136,E2 16912.136} C_VEL
LIN {X 0,Y 443.33,Z 894.863,A -85,B 0,C 180,E1 16920.924,E2 16920.924} C_VEL
LIN {X 0,Y 448.471,Z 905.549,A -85,B 0,C 180,E1 16930.543,E2 16930.543} C_VEL
LIN {X 0,Y 460.715,Z 925.428,A -85,B 0,C 180,E1 16938.819,E2 16938.819} C_VEL
LIN {X 0,Y 476.912,Z 957.401,A -85,B 0,C 180,E1 16946.644,E2 16946.644} C_VEL
LIN {X 0,Y 490.437,Z 995.228,A -85,B 0,C 180,E1 16953.061,E2 16953.061} C_VEL
LIN {X 0,Y 468.398,Z 1067.395,A -85,B 0,C 180,E1 16957.717,E2 16957.717} C_VEL
LIN {X 0,Y 444.128,Z 1129.239,A -85,B 0,C 180,E1 16964.142,E2 16964.142} C_VEL
LIN {X 0,Y 421.361,Z 1181.338,A -85,B 0,C 180,E1 16972.682,E2 16972.682} C_VEL
LIN {X 0,Y 405.391,Z 1219.877,A -85,B 0,C 180,E1 16982.693,E2 16982.693} C_VEL
LIN {X 0,Y 397.469,Z 1244.815,A -85,B 0,C 180,E1 16993.353,E2 16993.353} C_VEL
LIN {X 0,Y 395.34,Z 1255.934,A -85,B 0,C 180,E1 17002.275,E2 17002.275} C_VEL
LIN {X 0,Y 395.237,Z 1258.874,A -85,B 0,C 180,E1 17011.1,E2 17011.1} C_VEL
LIN {X 0,Y 395.719,Z 1252.678,A -85,B 0,C 180,E1 17021.058,E2 17021.058} C_VEL
LIN {X 0,Y 400.374,Z 1233.867,A -85,B 0,C 180,E1 17031.979,E2 17031.979} C_VEL
LIN {X 0,Y 413.616,Z 1199.448,A -85,B 0,C 180,E1 17043.09,E2 17043.09} C_VEL
LIN {X 0,Y 433.819,Z 1153.015,A -85,B 0,C 180,E1 17052.348,E2 17052.348} C_VEL
LIN {X 0,Y 457.617,Z 1096.217,A -85,B 0,C 180,E1 17059.55,E2 17059.55} C_VEL
LIN {X 0,Y 481.144,Z 1029.599,A -85,B 0,C 180,E1 17064.856,E2 17064.856} C_VEL
LIN {X 0,Y 490.078,Z 994.238,A -85,B 0,C 180,E1 17066.993,E2 17066.993} C_VEL
LIN {X 0,Y 474.702,Z 952.554,A -85,B 0,C 180,E1 17074.243,E2 17074.243} C_VEL
LIN {X 0,Y 458.104,Z 920.689,A -85,B 0,C 180,E1 17082.504,E2 17082.504} C_VEL
LIN {X 0,Y 446.642,Z 901.311,A -85,B 0,C 180,E1 17091.264,E2 17091.264} C_VEL
LIN {X 0,Y 443.183,Z 894.512,A -85,B 0,C 180,E1 17101.037,E2 17101.037} C_VEL
LIN {X 0,Y 449.364,Z 906.569,A -85,B 0,C 180,E1 17110.758,E2 17110.758} C_VEL
LIN {X 0,Y 463.127,Z 927.638,A -85,B 0,C 180,E1 17119.099,E2 17119.099} C_VEL
LIN {X 0,Y 481.931,Z 963.954,A -85,B 0,C 180,E1 17127.219,E2 17127.219} C_VEL
LIN {X 0,Y 493.523,Z 997.553,A -85,B 0,C 180,E1 17132.315,E2 17132.315} C_VEL
LIN {X 0,Y 473.594,Z 1067.013,A -85,B 0,C 180,E1 17136.128,E2 17136.128} C_VEL
LIN {X 0,Y 448.869,Z 1133.845,A -85,B 0,C 180,E1 17142.103,E2 17142.103} C_VEL
LIN {X 0,Y 425.174,Z 1191.125,A -85,B 0,C 180,E1 17150.292,E2 17150.292} C_VEL
LIN {X 0,Y 407.314,Z 1235.752,A -85,B 0,C 180,E1 17160.342,E2 17160.342} C_VEL
LIN {X 0,Y 397.945,Z 1265.317,A -85,B 0,C 180,E1 17171.08,E2 17171.08} C_VEL
LIN {X 0,Y 395.37,Z 1280.712,A -85,B 0,C 180,E1 17181.166,E2 17181.166} C_VEL
LIN {X 0,Y 395.109,Z 1284.818,A -85,B 0,C 180,E1 17191.101,E2 17191.101} C_VEL
LIN {X 0,Y 395.716,Z 1278.355,A -85,B 0,C 180,E1 17200.94,E2 17200.94} C_VEL
LIN {X 0,Y 399.397,Z 1259.122,A -85,B 0,C 180,E1 17211.694,E2 17211.694} C_VEL
LIN {X 0,Y 410.87,Z 1225.63,A -85,B 0,C 180,E1 17222.396,E2 17222.396} C_VEL
LIN {X 0,Y 421.759,Z 1199.506,A -85,B 0,C 180,E1 17228.144,E2 17228.144} C_VEL
LIN {X 0,Y 423.091,Z 1180.722,A -85,B 0,C 180,E1 17232.23,E2 17232.23} C_VEL
LIN {X 0,Y 447.966,Z 1122.477,A -85,B 0,C 180,E1 17239.916,E2 17239.916} C_VEL
LIN {X 0,Y 472.489,Z 1055.891,A -85,B 0,C 180,E1 17245.43,E2 17245.43} C_VEL
LIN {X 0,Y 488.41,Z 998.152,A -85,B 0,C 180,E1 17248.586,E2 17248.586} C_VEL
LIN {X 0,Y 471.725,Z 955.724,A -85,B 0,C 180,E1 17255.957,E2 17255.957} C_VEL
LIN {X 0,Y 455.011,Z 925.905,A -85,B 0,C 180,E1 17264.286,E2 17264.286} C_VEL
LIN {X 0,Y 444.786,Z 908.92,A -85,B 0,C 180,E1 17272.594,E2 17272.594} C_VEL
LIN {X 0,Y 441.918,Z 902.862,A -85,B 0,C 180,E1 17280.927,E2 17280.927} C_VEL
LIN {X 0,Y 446.853,Z 913.478,A -85,B 0,C 180,E1 17290.495,E2 17290.495} C_VEL
LIN {X 0,Y 458.792,Z 933.695,A -85,B 0,C 180,E1 17298.9,E2 17298.9} C_VEL
LIN {X 0,Y 474.594,Z 967.413,A -85,B 0,C 180,E1 17306.999,E2 17306.999} C_VEL
LIN {X 0,Y 484.887,Z 1001.479,A -85,B 0,C 180,E1 17312.631,E2 17312.631} C_VEL
LIN {X 0,Y 462.225,Z 1071.009,A -85,B 0,C 180,E1 17317.191,E2 17317.191} C_VEL
LIN {X 0,Y 437.1,Z 1132.521,A -85,B 0,C 180,E1 17323.759,E2 17323.759} C_VEL
LIN {X 0,Y 413.839,Z 1183.737,A -85,B 0,C 180,E1 17332.426,E2 17332.426} C_VEL
LIN {X 0,Y 397.433,Z 1221.847,A -85,B 0,C 180,E1 17342.717,E2 17342.717} C_VEL
LIN {X 0,Y 389.071,Z 1246.959,A -85,B 0,C 180,E1 17354.149,E2 17354.149} C_VEL
LIN {X 0,Y 387.201,Z 1257.735,A -85,B 0,C 180,E1 17364.374,E2 17364.374} C_VEL
LIN {X 0,Y 387.197,Z 1258.601,A -85,B 0,C 180,E1 17373.567,E2 17373.567} C_VEL
LIN {X 0,Y 388.273,Z 1250.121,A -85,B 0,C 180,E1 17383.567,E2 17383.567} C_VEL
LIN {X 0,Y 395,Z 1228.109,A -85,B 0,C 180,E1 17394.893,E2 17394.893} C_VEL
LIN {X 0,Y 410.634,Z 1190.725,A -85,B 0,C 180,E1 17405.913,E2 17405.913} C_VEL
LIN {X 0,Y 433.066,Z 1141.581,A -85,B 0,C 180,E1 17414.867,E2 17414.867} C_VEL
LIN {X 0,Y 458.498,Z 1080.582,A -85,B 0,C 180,E1 17421.879,E2 17421.879} C_VEL
LIN {X 0,Y 481.896,Z 1011.777,A -85,B 0,C 180,E1 17426.727,E2 17426.727} C_VEL
LIN {X 0,Y 484.666,Z 997.825,A -85,B 0,C 180,E1 17427.664,E2 17427.664} C_VEL
LIN {X 0,Y 469.719,Z 955.941,A -85,B 0,C 180,E1 17435.23,E2 17435.23} C_VEL
LIN {X 0,Y 454.367,Z 926.083,A -85,B 0,C 180,E1 17443.516,E2 17443.516} C_VEL
LIN {X 0,Y 444.67,Z 908.855,A -85,B 0,C 180,E1 17451.719,E2 17451.719} C_VEL
LIN {X 0,Y 441.809,Z 902.526,A -85,B 0,C 180,E1 17461.04,E2 17461.04} C_VEL
LIN {X 0,Y 447.854,Z 914.561,A -85,B 0,C 180,E1 17470.795,E2 17470.795} C_VEL
LIN {X 0,Y 460.852,Z 935.645,A -85,B 0,C 180,E1 17479.016,E2 17479.016} C_VEL
LIN {X 0,Y 478.168,Z 970.654,A -85,B 0,C 180,E1 17486.94,E2 17486.94} C_VEL
LIN {X 0,Y 488.45,Z 1000.531,A -85,B 0,C 180,E1 17491.645,E2 17491.645} C_VEL
LIN {X 0,Y 467.728,Z 1069.847,A -85,B 0,C 180,E1 17495.534,E2 17495.534} C_VEL
LIN {X 0,Y 442.439,Z 1135.702,A -85,B 0,C 180,E1 17501.545,E2 17501.545} C_VEL
LIN {X 0,Y 418.721,Z 1190.846,A -85,B 0,C 180,E1 17509.555,E2 17509.555} C_VEL
LIN {X 0,Y 399.984,Z 1235.688,A -85,B 0,C 180,E1 17519.809,E2 17519.809} C_VEL
LIN {X 0,Y 390.185,Z 1265.047,A -85,B 0,C 180,E1 17530.689,E2 17530.689} C_VEL
LIN {X 0,Y 387.382,Z 1280.446,A -85,B 0,C 180,E1 17540.982,E2 17540.982} C_VEL
LIN {X 0,Y 387.121,Z 1284.556,A -85,B 0,C 180,E1 17551.124,E2 17551.124} C_VEL
LIN {X 0,Y 387.755,Z 1278.224,A -85,B 0,C 180,E1 17561.046,E2 17561.046} C_VEL
LIN {X 0,Y 391.374,Z 1260.089,A -85,B 0,C 180,E1 17571.624,E2 17571.624} C_VEL
LIN {X 0,Y 402.687,Z 1228.251,A -85,B 0,C 180,E1 17582.302,E2 17582.302} C_VEL
LIN {X 0,Y 423.091,Z 1180.722,A -85,B 0,C 180,E1 17592.23,E2 17592.23} C_VEL
LIN {X 0,Y 426.135,Z 1160.121,A -85,B 0,C 180,E1 17596.116,E2 17596.116} C_VEL
LIN {X 0,Y 452.569,Z 1097.584,A -85,B 0,C 180,E1 17603.099,E2 17603.099} C_VEL
LIN {X 0,Y 476.274,Z 1029.162,A -85,B 0,C 180,E1 17607.796,E2 17607.796} C_VEL
LIN {X 0,Y 483.204,Z 1001.774,A -85,B 0,C 180,E1 17609.262,E2 17609.262} C_VEL
LIN {X 0,Y 467.342,Z 960.466,A -85,B 0,C 180,E1 17616.742,E2 17616.742} C_VEL
LIN {X 0,Y 450.911,Z 929.747,A -85,B 0,C 180,E1 17625.728,E2 17625.728} C_VEL
LIN {X 0,Y 442.251,Z 916.012,A -85,B 0,C 180,E1 17633.789,E2 17633.789} C_VEL
LIN {X 0,Y 440.362,Z 911.067,A -85,B 0,C 180,E1 17641.177,E2 17641.177} C_VEL
LIN {X 0,Y 444.976,Z 921.283,A -85,B 0,C 180,E1 17650.456,E2 17650.456} C_VEL
LIN {X 0,Y 456.715,Z 942.198,A -85,B 0,C 180,E1 17659.09,E2 17659.09} C_VEL
LIN {X 0,Y 471.564,Z 976.402,A -85,B 0,C 180,E1 17667.187,E2 17667.187} C_VEL
LIN {X 0,Y 479.424,Z 1006.016,A -85,B 0,C 180,E1 17672.036,E2 17672.036} C_VEL
LIN {X 0,Y 455.873,Z 1075.23,A -85,B 0,C 180,E1 17676.706,E2 17676.706} C_VEL
LIN {X 0,Y 429.439,Z 1137.141,A -85,B 0,C 180,E1 17683.555,E2 17683.555} C_VEL
LIN {X 0,Y 405.564,Z 1187.712,A -85,B 0,C 180,E1 17692.535,E2 17692.535} C_VEL
LIN {X 0,Y 388.84,Z 1225.324,A -85,B 0,C 180,E1 17703.321,E2 17703.321} C_VEL
LIN {X 0,Y 380.678,Z 1248.992,A -85,B 0,C 180,E1 17714.976,E2 17714.976} C_VEL
LIN {X 0,Y 379.204,Z 1257.999,A -85,B 0,C 180,E1 17724.255,E2 17724.255} C_VEL
LIN {X 0,Y 379.237,Z 1258.951,A -85,B 0,C 180,E1 17733.442,E2 17733.442} C_VEL
LIN {X 0,Y 380.382,Z 1250.389,A -85,B 0,C 180,E1 17743.854,E2 17743.854} C_VEL
LIN {X 0,Y 387.838,Z 1227.369,A -85,B 0,C 180,E1 17755.807,E2 17755.807} C_VEL
LIN {X 0,Y 404.498,Z 1189.655,A -85,B 0,C 180,E1 17766.928,E2 17766.928} C_VEL
LIN {X 0,Y 428.041,Z 1140.12,A -85,B 0,C 180,E1 17775.905,E2 17775.905} C_VEL
LIN {X 0,Y 453.689,Z 1080.372,A -85,B 0,C 180,E1 17782.736,E2 17782.736} C_VEL
LIN {X 0,Y 477.507,Z 1012.026,A -85,B 0,C 180,E1 17787.541,E2 17787.541} C_VEL
LIN {X 0,Y 479.344,Z 1001.43,A -85,B 0,C 180,E1 17788.345,E2 17788.345} C_VEL
LIN {X 0,Y 465.833,Z 962.008,A -85,B 0,C 180,E1 17795.685,E2 17795.685} C_VEL
LIN {X 0,Y 451.471,Z 932.534,A -85,B 0,C 180,E1 17804.095,E2 17804.095} C_VEL
LIN {X 0,Y 442.693,Z 916.43,A -85,B 0,C 180,E1 17812.178,E2 17812.178} C_VEL
LIN {X 0,Y 440.274,Z 910.502,A -85,B 0,C 180,E1 17821.044,E2 17821.044} C_VEL
LIN {X 0,Y 446.248,Z 922.562,A -85,B 0,C 180,E1 17830.834,E2 17830.834} C_VEL
LIN {X 0,Y 458.985,Z 944.481,A -85,B 0,C 180,E1 17839.184,E2 17839.184} C_VEL
LIN {X 0,Y 475.113,Z 979.174,A -85,B 0,C 180,E1 17846.985,E2 17846.985} C_VEL
LIN {X 0,Y 483.057,Z 1004.93,A -85,B 0,C 180,E1 17851.027,E2 17851.027} C_VEL
LIN {X 0,Y 461.885,Z 1072.703,A -85,B 0,C 180,E1 17854.923,E2 17854.923} C_VEL
LIN {X 0,Y 435.525,Z 1138.817,A -85,B 0,C 180,E1 17861.116,E2 17861.116} C_VEL
LIN {X 0,Y 410.284,Z 1195.226,A -85,B 0,C 180,E1 17869.645,E2 17869.645} C_VEL
LIN {X 0,Y 391.142,Z 1239.245,A -85,B 0,C 180,E1 17880.34,E2 17880.34} C_VEL
LIN {X 0,Y 381.437,Z 1268.184,A -85,B 0,C 180,E1 17892.035,E2 17892.035} C_VEL
LIN {X 0,Y 379.36,Z 1281.086,A -85,B 0,C 180,E1 17901.949,E2 17901.949} C_VEL
LIN {X 0,Y 379.12,Z 1284.293,A -85,B 0,C 180,E1 17911.148,E2 17911.148} C_VEL
LIN {X 0,Y 379.804,Z 1277.694,A -85,B 0,C 180,E1 17921.525,E2 17921.525} C_VEL
LIN {X 0,Y 383.975,Z 1258.437,A -85,B 0,C 180,E1 17932.675,E2 17932.675} C_VEL
LIN {X 0,Y 396.167,Z 1226.382,A -85,B 0,C 180,E1 17943.369,E2 17943.369} C_VEL
LIN {X 0,Y 417.433,Z 1179.186,A -85,B 0,C 180,E1 17953.215,E2 17953.215} C_VEL
LIN {X 0,Y 426.135,Z 1160.121,A -85,B 0,C 180,E1 17956.116,E2 17956.116} C_VEL
LIN {X 0,Y 430.384,Z 1137.999,A -85,B 0,C 180,E1 17959.789,E2 17959.789} C_VEL
LIN {X 0,Y 457.2,Z 1072.235,A -85,B 0,C 180,E1 17965.974,E2 17965.974} C_VEL
LIN {X 0,Y 477.976,Z 1005.625,A -85,B 0,C 180,E1 17969.918,E2 17969.918} C_VEL
LIN {X 0,Y 463.386,Z 966.07,A -85,B 0,C 180,E1 17977.316,E2 17977.316} C_VEL
LIN {X 0,Y 448.11,Z 936.579,A -85,B 0,C 180,E1 17986.278,E2 17986.278} C_VEL
LIN {X 0,Y 440.282,Z 923.586,A -85,B 0,C 180,E1 17994.133,E2 17994.133} C_VEL
LIN {X 0,Y 438.744,Z 919.14,A -85,B 0,C 180,E1 18001.305,E2 18001.305} C_VEL
LIN {X 0,Y 442.985,Z 929.073,A -85,B 0,C 180,E1 18010.386,E2 18010.386} C_VEL
LIN {X 0,Y 454.035,Z 949.846,A -85,B 0,C 180,E1 18018.956,E2 18018.956} C_VEL
LIN {X 0,Y 467.641,Z 983.247,A -85,B 0,C 180,E1 18026.953,E2 18026.953} C_VEL
LIN {X 0,Y 474.484,Z 1008.525,A -85,B 0,C 180,E1 18031.332,E2 18031.332} C_VEL
LIN {X 0,Y 450.007,Z 1077.914,A -85,B 0,C 180,E1 18036.089,E2 18036.089} C_VEL
LIN {X 0,Y 422.849,Z 1139.275,A -85,B 0,C 180,E1 18043.015,E2 18043.015} C_VEL
LIN {X 0,Y 398.362,Z 1189.163,A -85,B 0,C 180,E1 18052.083,E2 18052.083} C_VEL
LIN {X 0,Y 380.841,Z 1226.97,A -85,B 0,C 180,E1 18063.302,E2 18063.302} C_VEL
LIN {X 0,Y 372.826,Z 1249.259,A -85,B 0,C 180,E1 18074.652,E2 18074.652} C_VEL
LIN {X 0,Y 371.227,Z 1258.262,A -85,B 0,C 180,E1 18084.131,E2 18084.131} C_VEL
LIN {X 0,Y 371.248,Z 1259.214,A -85,B 0,C 180,E1 18093.516,E2 18093.516} C_VEL
LIN {X 0,Y 372.512,Z 1250.656,A -85,B 0,C 180,E1 18104.153,E2 18104.153} C_VEL
LIN {X 0,Y 380.351,Z 1227.729,A -85,B 0,C 180,E1 18116.316,E2 18116.316} C_VEL
LIN {X 0,Y 397.806,Z 1190.014,A -85,B 0,C 180,E1 18127.632,E2 18127.632} C_VEL
LIN {X 0,Y 422.298,Z 1140.396,A -85,B 0,C 180,E1 18136.715,E2 18136.715} C_VEL
LIN {X 0,Y 449.152,Z 1079.832,A -85,B 0,C 180,E1 18143.635,E2 18143.635} C_VEL
LIN {X 0,Y 473.946,Z 1009.893,A -85,B 0,C 180,E1 18148.503,E2 18148.503} C_VEL
LIN {X 0,Y 466.17,Z 979.336,A -85,B 0,C 180,E1 18153.72,E2 18153.72} C_VEL
LIN {X 0,Y 452.403,Z 946.913,A -85,B 0,C 180,E1 18161.862,E2 18161.862} C_VEL
LIN {X 0,Y 441.502,Z 924.671,A -85,B 0,C 180,E1 18171.41,E2 18171.41} C_VEL
LIN {X 0,Y 438.718,Z 918.479,A -85,B 0,C 180,E1 18181.048,E2 18181.048} C_VEL
LIN {X 0,Y 445.085,Z 931.153,A -85,B 0,C 180,E1 18191.423,E2 18191.423} C_VEL
LIN {X 0,Y 458.842,Z 957.062,A -85,B 0,C 180,E1 18200.437,E2 18200.437} C_VEL
LIN {X 0,Y 474.585,Z 995.259,A -85,B 0,C 180,E1 18208.397,E2 18208.397} C_VEL
LIN {X 0,Y 477.348,Z 1010.076,A -85,B 0,C 180,E1 18210.438,E2 18210.438} C_VEL
LIN {X 0,Y 455.283,Z 1077.706,A -85,B 0,C 180,E1 18214.468,E2 18214.468} C_VEL
LIN {X 0,Y 428.367,Z 1142.265,A -85,B 0,C 180,E1 18220.727,E2 18220.727} C_VEL
LIN {X 0,Y 402.529,Z 1197.659,A -85,B 0,C 180,E1 18229.416,E2 18229.416} C_VEL
LIN {X 0,Y 383.076,Z 1240.75,A -85,B 0,C 180,E1 18240.307,E2 18240.307} C_VEL
LIN {X 0,Y 373.641,Z 1267.914,A -85,B 0,C 180,E1 18251.647,E2 18251.647} C_VEL
LIN {X 0,Y 371.371,Z 1280.821,A -85,B 0,C 180,E1 18261.775,E2 18261.775} C_VEL
LIN {X 0,Y 371.119,Z 1284.03,A -85,B 0,C 180,E1 18271.173,E2 18271.173} C_VEL
LIN {X 0,Y 371.819,Z 1277.426,A -85,B 0,C 180,E1 18281.776,E2 18281.776} C_VEL
LIN {X 0,Y 376.325,Z 1258.165,A -85,B 0,C 180,E1 18293.162,E2 18293.162} C_VEL
LIN {X 0,Y 389.265,Z 1225.864,A -85,B 0,C 180,E1 18304.115,E2 18304.115} C_VEL
LIN {X 0,Y 411.602,Z 1178.284,A -85,B 0,C 180,E1 18314.124,E2 18314.124} C_VEL
LIN {X 0,Y 430.384,Z 1137.999,A -85,B 0,C 180,E1 18319.789,E2 18319.789} C_VEL
LIN {X 0,Y 435.54,Z 1114.2,A -85,B 0,C 180,E1 18323.212,E2 18323.212} C_VEL
LIN {X 0,Y 461.183,Z 1048.683,A -85,B 0,C 180,E1 18328.352,E2 18328.352} C_VEL
LIN {X 0,Y 472.973,Z 1010.292,A -85,B 0,C 180,E1 18330.448,E2 18330.448} C_VEL
LIN {X 0,Y 459.007,Z 970.632,A -85,B 0,C 180,E1 18338.111,E2 18338.111} C_VEL
LIN {X 0,Y 444.862,Z 942.741,A -85,B 0,C 180,E1 18347.135,E2 18347.135} C_VEL
LIN {X 0,Y 438.184,Z 931.106,A -85,B 0,C 180,E1 18354.479,E2 18354.479} C_VEL
LIN {X 0,Y 436.851,Z 927.103,A -85,B 0,C 180,E1 18361.435,E2 18361.435} C_VEL
LIN {X 0,Y 441.017,Z 936.999,A -85,B 0,C 180,E1 18370.433,E2 18370.433} C_VEL
LIN {X 0,Y 450.812,Z 956.579,A -85,B 0,C 180,E1 18378.587,E2 18378.587} C_VEL
LIN {X 0,Y 463.395,Z 989.061,A -85,B 0,C 180,E1 18386.526,E2 18386.526} C_VEL
LIN {X 0,Y 468.797,Z 1013.676,A -85,B 0,C 180,E1 18390.762,E2 18390.762} C_VEL
LIN {X 0,Y 443.513,Z 1082.265,A -85,B 0,C 180,E1 18395.614,E2 18395.614} C_VEL
LIN {X 0,Y 415.641,Z 1142.633,A -85,B 0,C 180,E1 18402.633,E2 18402.633} C_VEL
LIN {X 0,Y 390.621,Z 1191.796,A -85,B 0,C 180,E1 18411.904,E2 18411.904} C_VEL
LIN {X 0,Y 373.035,Z 1228.157,A -85,B 0,C 180,E1 18423.098,E2 18423.098} C_VEL
LIN {X 0,Y 364.983,Z 1249.525,A -85,B 0,C 180,E1 18434.313,E2 18434.313} C_VEL
LIN {X 0,Y 363.229,Z 1258.525,A -85,B 0,C 180,E1 18444.002,E2 18444.002} C_VEL
LIN {X 0,Y 363.241,Z 1259.477,A -85,B 0,C 180,E1 18453.594,E2 18453.594} C_VEL
LIN {X 0,Y 364.653,Z 1250.922,A -85,B 0,C 180,E1 18464.464,E2 18464.464} C_VEL
LIN {X 0,Y 372.888,Z 1228.005,A -85,B 0,C 180,E1 18476.885,E2 18476.885} C_VEL
LIN {X 0,Y 391.204,Z 1190.291,A -85,B 0,C 180,E1 18488.381,E2 18488.381} C_VEL
LIN {X 0,Y 417.042,Z 1139.931,A -85,B 0,C 180,E1 18497.653,E2 18497.653} C_VEL
LIN {X 0,Y 444.071,Z 1080.734,A -85,B 0,C 180,E1 18504.43,E2 18504.43} C_VEL
LIN {X 0,Y 469.093,Z 1010.163,A -85,B 0,C 180,E1 18509.49,E2 18509.49} C_VEL
LIN {X 0,Y 457.028,Z 971.328,A -85,B 0,C 180,E1 18517.258,E2 18517.258} C_VEL
LIN {X 0,Y 444.422,Z 943.538,A -85,B 0,C 180,E1 18526.001,E2 18526.001} C_VEL
LIN {X 0,Y 438.125,Z 931.315,A -85,B 0,C 180,E1 18533.236,E2 18533.236} C_VEL
LIN {X 0,Y 436.839,Z 926.22,A -85,B 0,C 180,E1 18540.928,E2 18540.928} C_VEL
LIN {X 0,Y 443.227,Z 939.058,A -85,B 0,C 180,E1 18551.471,E2 18551.471} C_VEL
LIN {X 0,Y 456.322,Z 965.261,A -85,B 0,C 180,E1 18560.491,E2 18560.491} C_VEL
LIN {X 0,Y 471.31,Z 1004.578,A -85,B 0,C 180,E1 18568.613,E2 18568.613} C_VEL
LIN {X 0,Y 472.188,Z 1013.53,A -85,B 0,C 180,E1 18569.758,E2 18569.758} C_VEL
LIN {X 0,Y 448.636,Z 1082.503,A -85,B 0,C 180,E1 18574,E2 18574} C_VEL
LIN {X 0,Y 420.332,Z 1147.409,A -85,B 0,C 180,E1 18580.557,E2 18580.557} C_VEL
LIN {X 0,Y 393.921,Z 1201.814,A -85,B 0,C 180,E1 18589.533,E2 18589.533} C_VEL
LIN {X 0,Y 374.969,Z 1242.328,A -85,B 0,C 180,E1 18600.295,E2 18600.295} C_VEL
LIN {X 0,Y 365.518,Z 1268.639,A -85,B 0,C 180,E1 18611.851,E2 18611.851} C_VEL
LIN {X 0,Y 363.368,Z 1280.555,A -85,B 0,C 180,E1 18621.592,E2 18621.592} C_VEL
LIN {X 0,Y 363.117,Z 1283.768,A -85,B 0,C 180,E1 18631.199,E2 18631.199} C_VEL
LIN {X 0,Y 363.839,Z 1277.281,A -85,B 0,C 180,E1 18641.92,E2 18641.92} C_VEL
LIN {X 0,Y 368.227,Z 1259.27,A -85,B 0,C 180,E1 18653.059,E2 18653.059} C_VEL
LIN {X 0,Y 381.279,Z 1227.85,A -85,B 0,C 180,E1 18664.223,E2 18664.223} C_VEL
LIN {X 0,Y 404.072,Z 1181.273,A -85,B 0,C 180,E1 18674.41,E2 18674.41} C_VEL
LIN {X 0,Y 432.12,Z 1122.091,A -85,B 0,C 180,E1 18682.406,E2 18682.406} C_VEL
LIN {X 0,Y 435.54,Z 1114.2,A -85,B 0,C 180,E1 18683.212,E2 18683.212} C_VEL
LIN {X 0,Y 441.293,Z 1088.931,A -85,B 0,C 180,E1 18686.389,E2 18686.389} C_VEL
LIN {X 0,Y 467.033,Z 1017.669,A -85,B 0,C 180,E1 18690.903,E2 18690.903} C_VEL
LIN {X 0,Y 465.102,Z 1004.32,A -85,B 0,C 180,E1 18692.832,E2 18692.832} C_VEL
LIN {X 0,Y 452.234,Z 970.173,A -85,B 0,C 180,E1 18700.339,E2 18700.339} C_VEL
LIN {X 0,Y 439.974,Z 945.503,A -85,B 0,C 180,E1 18709.582,E2 18709.582} C_VEL
LIN {X 0,Y 435.146,Z 934.543,A -85,B 0,C 180,E1 18718.944,E2 18718.944} C_VEL
LIN {X 0,Y 437.973,Z 943.226,A -85,B 0,C 180,E1 18729.472,E2 18729.472} C_VEL
LIN {X 0,Y 447.501,Z 963.292,A -85,B 0,C 180,E1 18738.218,E2 18738.218} C_VEL
LIN {X 0,Y 459.397,Z 996.344,A -85,B 0,C 180,E1 18746.417,E2 18746.417} C_VEL
LIN {X 0,Y 463.701,Z 1017.071,A -85,B 0,C 180,E1 18750.077,E2 18750.077} C_VEL
LIN {X 0,Y 437.892,Z 1084.599,A -85,B 0,C 180,E1 18754.933,E2 18754.933} C_VEL
LIN {X 0,Y 408.871,Z 1145.255,A -85,B 0,C 180,E1 18762.133,E2 18762.133} C_VEL
LIN {X 0,Y 383.44,Z 1193.294,A -85,B 0,C 180,E1 18771.435,E2 18771.435} C_VEL
LIN {X 0,Y 365.675,Z 1228.421,A -85,B 0,C 180,E1 18782.508,E2 18782.508} C_VEL
LIN {X 0,Y 357.154,Z 1249.792,A -85,B 0,C 180,E1 18793.96,E2 18793.96} C_VEL
LIN {X 0,Y 355.231,Z 1258.789,A -85,B 0,C 180,E1 18803.866,E2 18803.866} C_VEL
LIN {X 0,Y 355.257,Z 1259.74,A -85,B 0,C 180,E1 18813.674,E2 18813.674} C_VEL
LIN {X 0,Y 356.781,Z 1251.19,A -85,B 0,C 180,E1 18824.791,E2 18824.791} C_VEL
LIN {X 0,Y 365.515,Z 1228.217,A -85,B 0,C 180,E1 18837.5,E2 18837.5} C_VEL
LIN {X 0,Y 384.676,Z 1190.621,A -85,B 0,C 180,E1 18849.139,E2 18849.139} C_VEL
LIN {X 0,Y 411.481,Z 1140.208,A -85,B 0,C 180,E1 18858.509,E2 18858.509} C_VEL
LIN {X 0,Y 439.655,Z 1080.322,A -85,B 0,C 180,E1 18865.361,E2 18865.361} C_VEL
LIN {X 0,Y 463.868,Z 1014.112,A -85,B 0,C 180,E1 18870.142,E2 18870.142} C_VEL
LIN {X 0,Y 452.513,Z 975.872,A -85,B 0,C 180,E1 18878.091,E2 18878.091} C_VEL
LIN {X 0,Y 440.886,Z 949.103,A -85,B 0,C 180,E1 18887.07,E2 18887.07} C_VEL
LIN {X 0,Y 435.879,Z 938.758,A -85,B 0,C 180,E1 18893.625,E2 18893.625} C_VEL
LIN {X 0,Y 434.95,Z 934.102,A -85,B 0,C 180,E1 18900.932,E2 18900.932} C_VEL
LIN {X 0,Y 440.815,Z 946.659,A -85,B 0,C 180,E1 18911.323,E2 18911.323} C_VEL
LIN {X 0,Y 452.857,Z 971.911,A -85,B 0,C 180,E1 18920.143,E2 18920.143} C_VEL
LIN {X 0,Y 466.608,Z 1010.034,A -85,B 0,C 180,E1 18928.191,E2 18928.191} C_VEL
LIN {X 0,Y 466.601,Z 1018.671,A -85,B 0,C 180,E1 18929.141,E2 18929.141} C_VEL
LIN {X 0,Y 442.192,Z 1086.828,A -85,B 0,C 180,E1 18933.478,E2 18933.478} C_VEL
LIN {X 0,Y 413.724,Z 1149.624,A -85,B 0,C 180,E1 18940.001,E2 18940.001} C_VEL
LIN {X 0,Y 386.809,Z 1202.963,A -85,B 0,C 180,E1 18949.022,E2 18949.022} C_VEL
LIN {X 0,Y 367.079,Z 1243.443,A -85,B 0,C 180,E1 18960.125,E2 18960.125} C_VEL
LIN {X 0,Y 357.72,Z 1268.369,A -85,B 0,C 180,E1 18971.441,E2 18971.441} C_VEL
LIN {X 0,Y 355.384,Z 1280.29,A -85,B 0,C 180,E1 18981.402,E2 18981.402} C_VEL
LIN {X 0,Y 355.131,Z 1283.506,A -85,B 0,C 180,E1 18991.225,E2 18991.225} C_VEL
LIN {X 0,Y 355.883,Z 1276.888,A -85,B 0,C 180,E1 19002.316,E2 19002.316} C_VEL
LIN {X 0,Y 361.012,Z 1257.837,A -85,B 0,C 180,E1 19014.102,E2 19014.102} C_VEL
LIN {X 0,Y 375.41,Z 1225.365,A -85,B 0,C 180,E1 19025.544,E2 19025.544} C_VEL
LIN {X 0,Y 399.734,Z 1177.75,A -85,B 0,C 180,E1 19035.795,E2 19035.795} C_VEL
LIN {X 0,Y 428.185,Z 1119.325,A -85,B 0,C 180,E1 19043.55,E2 19043.55} C_VEL
LIN {X 0,Y 441.293,Z 1088.931,A -85,B 0,C 180,E1 19046.389,E2 19046.389} C_VEL
LIN {X 0,Y 447.608,Z 1062.008,A -85,B 0,C 180,E1 19049.252,E2 19049.252} C_VEL
LIN {X 0,Y 462.315,Z 1016.599,A -85,B 0,C 180,E1 19052.057,E2 19052.057} C_VEL
LIN {X 0,Y 450.426,Z 980.255,A -85,B 0,C 180,E1 19059.721,E2 19059.721} C_VEL
LIN {X 0,Y 437.914,Z 953.509,A -85,B 0,C 180,E1 19069.388,E2 19069.388} C_VEL
LIN {X 0,Y 432.981,Z 943.784,A -85,B 0,C 180,E1 19077.755,E2 19077.755} C_VEL
LIN {X 0,Y 432.867,Z 944.406,A -85,B 0,C 180,E1 19083.459,E2 19083.459} C_VEL
LIN {X 0,Y 436.98,Z 953.222,A -85,B 0,C 180,E1 19090.951,E2 19090.951} C_VEL
LIN {X 0,Y 447.01,Z 977.252,A -85,B 0,C 180,E1 19100.055,E2 19100.055} C_VEL
LIN {X 0,Y 457.768,Z 1013.127,A -85,B 0,C 180,E1 19108.186,E2 19108.186} C_VEL
LIN {X 0,Y 458.04,Z 1022.414,A -85,B 0,C 180,E1 19109.485,E2 19109.485} C_VEL
LIN {X 0,Y 431.421,Z 1089.064,A -85,B 0,C 180,E1 19114.437,E2 19114.437} C_VEL
LIN {X 0,Y 401.664,Z 1148.792,A -85,B 0,C 180,E1 19121.757,E2 19121.757} C_VEL
LIN {X 0,Y 375.05,Z 1197.197,A -85,B 0,C 180,E1 19131.553,E2 19131.553} C_VEL
LIN {X 0,Y 356.532,Z 1232.399,A -85,B 0,C 180,E1 19143.442,E2 19143.442} C_VEL
LIN {X 0,Y 348.331,Z 1253.094,A -85,B 0,C 180,E1 19156.13,E2 19156.13} C_VEL
LIN {X 0,Y 347.21,Z 1260.043,A -85,B 0,C 180,E1 19166.239,E2 19166.239} C_VEL
LIN {X 0,Y 347.214,Z 1259.015,A -85,B 0,C 180,E1 19176.275,E2 19176.275} C_VEL
LIN {X 0,Y 350.167,Z 1247.534,A -85,B 0,C 180,E1 19188.101,E2 19188.101} C_VEL
LIN {X 0,Y 361.229,Z 1221.956,A -85,B 0,C 180,E1 19200.705,E2 19200.705} C_VEL
LIN {X 0,Y 383.082,Z 1182.106,A -85,B 0,C 180,E1 19211.969,E2 19211.969} C_VEL
LIN {X 0,Y 411.723,Z 1129.45,A -85,B 0,C 180,E1 19220.92,E2 19220.92} C_VEL
LIN {X 0,Y 440.529,Z 1068.052,A -85,B 0,C 180,E1 19227.288,E2 19227.288} C_VEL
LIN {X 0,Y 458.693,Z 1017.942,A -85,B 0,C 180,E1 19230.829,E2 19230.829} C_VEL
LIN {X 0,Y 448.164,Z 980.755,A -85,B 0,C 180,E1 19238.868,E2 19238.868} C_VEL
LIN {X 0,Y 437.65,Z 954.624,A -85,B 0,C 180,E1 19248.053,E2 19248.053} C_VEL
LIN {X 0,Y 433.198,Z 945.794,A -85,B 0,C 180,E1 19254.531,E2 19254.531} C_VEL
LIN {X 0,Y 432.87,Z 941.941,A -85,B 0,C 180,E1 19260.936,E2 19260.936} C_VEL
LIN {X 0,Y 438.319,Z 954.247,A -85,B 0,C 180,E1 19271.159,E2 19271.159} C_VEL
LIN {X 0,Y 450.497,Z 981.221,A -85,B 0,C 180,E1 19280.478,E2 19280.478} C_VEL
LIN {X 0,Y 462.563,Z 1018.05,A -85,B 0,C 180,E1 19288.193,E2 19288.193} C_VEL
LIN {X 0,Y 437.49,Z 1087.074,A -85,B 0,C 180,E1 19292.62,E2 19292.62} C_VEL
LIN {X 0,Y 408.401,Z 1149.347,A -85,B 0,C 180,E1 19299.103,E2 19299.103} C_VEL
LIN {X 0,Y 380.184,Z 1203.251,A -85,B 0,C 180,E1 19308.31,E2 19308.31} C_VEL
LIN {X 0,Y 359.284,Z 1244.357,A -85,B 0,C 180,E1 19319.876,E2 19319.876} C_VEL
LIN {X 0,Y 349.49,Z 1269.5,A -85,B 0,C 180,E1 19331.911,E2 19331.911} C_VEL
LIN {X 0,Y 347.149,Z 1281.688,A -85,B 0,C 180,E1 19343.724,E2 19343.724} C_VEL
LIN {X 0,Y 347.129,Z 1283.243,A -85,B 0,C 180,E1 19351.254,E2 19351.254} C_VEL
LIN {X 0,Y 347.932,Z 1276.621,A -85,B 0,C 180,E1 19362.602,E2 19362.602} C_VEL
LIN {X 0,Y 353.379,Z 1257.657,A -85,B 0,C 180,E1 19374.612,E2 19374.612} C_VEL
LIN {X 0,Y 369.261,Z 1223.984,A -85,B 0,C 180,E1 19386.594,E2 19386.594} C_VEL
LIN {X 0,Y 394.758,Z 1175.846,A -85,B 0,C 180,E1 19396.944,E2 19396.944} C_VEL
LIN {X 0,Y 424.428,Z 1116.566,A -85,B 0,C 180,E1 19404.712,E2 19404.712} C_VEL
LIN {X 0,Y 447.608,Z 1062.008,A -85,B 0,C 180,E1 19409.252,E2 19409.252} C_VEL
LIN {X 0,Y 453.859,Z 1033.617,A -85,B 0,C 180,E1 19411.844,E2 19411.844} C_VEL
LIN {X 0,Y 457.39,Z 1020.971,A -85,B 0,C 180,E1 19412.68,E2 19412.68} C_VEL
LIN {X 0,Y 446.767,Z 986.902,A -85,B 0,C 180,E1 19420.042,E2 19420.042} C_VEL
LIN {X 0,Y 435.949,Z 962.286,A -85,B 0,C 180,E1 19428.907,E2 19428.907} C_VEL
LIN {X 0,Y 431.027,Z 952.902,A -85,B 0,C 180,E1 19436.284,E2 19436.284} C_VEL
LIN {X 0,Y 430.57,Z 950.961,A -85,B 0,C 180,E1 19442.086,E2 19442.086} C_VEL
LIN {X 0,Y 434.428,Z 961.084,A -85,B 0,C 180,E1 19451.016,E2 19451.016} C_VEL
LIN {X 0,Y 444.072,Z 985.856,A -85,B 0,C 180,E1 19460.279,E2 19460.279} C_VEL
LIN {X 0,Y 453.675,Z 1021.954,A -85,B 0,C 180,E1 19468.393,E2 19468.393} C_VEL
LIN {X 0,Y 425.699,Z 1091.836,A -85,B 0,C 180,E1 19473.76,E2 19473.76} C_VEL
LIN {X 0,Y 395.438,Z 1150.496,A -85,B 0,C 180,E1 19481.085,E2 19481.085} C_VEL
LIN {X 0,Y 368.039,Z 1198.351,A -85,B 0,C 180,E1 19490.978,E2 19490.978} C_VEL
LIN {X 0,Y 349.174,Z 1232.669,A -85,B 0,C 180,E1 19502.837,E2 19502.837} C_VEL
LIN {X 0,Y 340.437,Z 1253.361,A -85,B 0,C 180,E1 19515.802,E2 19515.802} C_VEL
LIN {X 0,Y 339.21,Z 1260.306,A -85,B 0,C 180,E1 19526.15,E2 19526.15} C_VEL
LIN {X 0,Y 339.223,Z 1259.28,A -85,B 0,C 180,E1 19536.423,E2 19536.423} C_VEL
LIN {X 0,Y 342.322,Z 1247.893,A -85,B 0,C 180,E1 19548.468,E2 19548.468} C_VEL
LIN {X 0,Y 354.129,Z 1222.23,A -85,B 0,C 180,E1 19561.389,E2 19561.389} C_VEL
LIN {X 0,Y 376.976,Z 1182.38,A -85,B 0,C 180,E1 19572.809,E2 19572.809} C_VEL
LIN {X 0,Y 406.995,Z 1128.952,A -85,B 0,C 180,E1 19581.924,E2 19581.924} C_VEL
LIN {X 0,Y 436.4,Z 1067.822,A -85,B 0,C 180,E1 19588.228,E2 19588.228} C_VEL
LIN {X 0,Y 453.449,Z 1021.395,A -85,B 0,C 180,E1 19591.614,E2 19591.614} C_VEL
LIN {X 0,Y 443.96,Z 985.843,A -85,B 0,C 180,E1 19599.608,E2 19599.608} C_VEL
LIN {X 0,Y 434.257,Z 960.566,A -85,B 0,C 180,E1 19608.98,E2 19608.98} C_VEL
LIN {X 0,Y 430.536,Z 952.592,A -85,B 0,C 180,E1 19615.764,E2 19615.764} C_VEL
LIN {X 0,Y 430.62,Z 949.752,A -85,B 0,C 180,E1 19620.941,E2 19620.941} C_VEL
LIN {X 0,Y 434.88,Z 960.399,A -85,B 0,C 180,E1 19630.104,E2 19630.104} C_VEL
LIN {X 0,Y 445.127,Z 983.478,A -85,B 0,C 180,E1 19638.952,E2 19638.952} C_VEL
LIN {X 0,Y 456.861,Z 1019.587,A -85,B 0,C 180,E1 19647.06,E2 19647.06} C_VEL
LIN {X 0,Y 455.218,Z 1029.032,A -85,B 0,C 180,E1 19647.902,E2 19647.902} C_VEL
LIN {X 0,Y 428.216,Z 1097.693,A -85,B 0,C 180,E1 19652.608,E2 19652.608} C_VEL
LIN {X 0,Y 397.281,Z 1160.188,A -85,B 0,C 180,E1 19659.734,E2 19659.734} C_VEL
LIN {X 0,Y 369.145,Z 1211.378,A -85,B 0,C 180,E1 19669.395,E2 19669.395} C_VEL
LIN {X 0,Y 349.213,Z 1249.749,A -85,B 0,C 180,E1 19681.433,E2 19681.433} C_VEL
LIN {X 0,Y 341,Z 1271.871,A -85,B 0,C 180,E1 19693.308,E2 19693.308} C_VEL
LIN {X 0,Y 339.173,Z 1281.424,A -85,B 0,C 180,E1 19703.576,E2 19703.576} C_VEL
LIN {X 0,Y 339.141,Z 1282.981,A -85,B 0,C 180,E1 19711.283,E2 19711.283} C_VEL
LIN {X 0,Y 339.966,Z 1276.353,A -85,B 0,C 180,E1 19722.902,E2 19722.902} C_VEL
LIN {X 0,Y 345.963,Z 1257.013,A -85,B 0,C 180,E1 19735.363,E2 19735.363} C_VEL
LIN {X 0,Y 363.168,Z 1222.6,A -85,B 0,C 180,E1 19747.688,E2 19747.688} C_VEL
LIN {X 0,Y 389.931,Z 1174.02,A -85,B 0,C 180,E1 19758.106,E2 19758.106} C_VEL
LIN {X 0,Y 420.554,Z 1114.445,A -85,B 0,C 180,E1 19765.828,E2 19765.828} C_VEL
LIN {X 0,Y 448.295,Z 1049.221,A -85,B 0,C 180,E1 19770.942,E2 19770.942} C_VEL
LIN {X 0,Y 453.859,Z 1033.617,A -85,B 0,C 180,E1 19771.844,E2 19771.844} C_VEL
LIN {X 0,Y 452.347,Z 1023.026,A -85,B 0,C 180,E1 19773.619,E2 19773.619} C_VEL
LIN {X 0,Y 451.123,Z 1020.029,A -85,B 0,C 180,E1 19774.325,E2 19774.325} C_VEL
LIN {X 0,Y 441.11,Z 988.799,A -85,B 0,C 180,E1 19781.789,E2 19781.789} C_VEL
LIN {X 0,Y 431.612,Z 966.822,A -85,B 0,C 180,E1 19790.84,E2 19790.84} C_VEL
LIN {X 0,Y 428.445,Z 957.677,A -85,B 0,C 180,E1 19800.956,E2 19800.956} C_VEL
LIN {X 0,Y 431.043,Z 967.334,A -85,B 0,C 180,E1 19810.077,E2 19810.077} C_VEL
LIN {X 0,Y 439.405,Z 989.528,A -85,B 0,C 180,E1 19819.088,E2 19819.088} C_VEL
LIN {X 0,Y 448.071,Z 1023.043,A -85,B 0,C 180,E1 19827.139,E2 19827.139} C_VEL
LIN {X 0,Y 447.599,Z 1030.191,A -85,B 0,C 180,E1 19828.114,E2 19828.114} C_VEL
LIN {X 0,Y 418.68,Z 1097.121,A -85,B 0,C 180,E1 19833.337,E2 19833.337} C_VEL
LIN {X 0,Y 387.605,Z 1154.803,A -85,B 0,C 180,E1 19840.84,E2 19840.84} C_VEL
LIN {X 0,Y 360.647,Z 1200.129,A -85,B 0,C 180,E1 19850.574,E2 19850.574} C_VEL
LIN {X 0,Y 341.03,Z 1234.335,A -85,B 0,C 180,E1 19862.897,E2 19862.897} C_VEL
LIN {X 0,Y 332.557,Z 1253.627,A -85,B 0,C 180,E1 19875.458,E2 19875.458} C_VEL
LIN {X 0,Y 331.205,Z 1260.569,A -85,B 0,C 180,E1 19886.057,E2 19886.057} C_VEL
LIN {X 0,Y 331.234,Z 1259.544,A -85,B 0,C 180,E1 19896.579,E2 19896.579} C_VEL
LIN {X 0,Y 334.564,Z 1248.014,A -85,B 0,C 180,E1 19909.023,E2 19909.023} C_VEL
LIN {X 0,Y 347.019,Z 1222.559,A -85,B 0,C 180,E1 19922.085,E2 19922.085} C_VEL
LIN {X 0,Y 370.71,Z 1182.978,A -85,B 0,C 180,E1 19933.613,E2 19933.613} C_VEL
LIN {X 0,Y 401.836,Z 1129.431,A -85,B 0,C 180,E1 19942.824,E2 19942.824} C_VEL
LIN {X 0,Y 432.165,Z 1068.12,A -85,B 0,C 180,E1 19949.141,E2 19949.141} C_VEL
LIN {X 0,Y 448.437,Z 1025.677,A -85,B 0,C 180,E1 19952.257,E2 19952.257} C_VEL
LIN {X 0,Y 439.752,Z 990.902,A -85,B 0,C 180,E1 19960.386,E2 19960.386} C_VEL
LIN {X 0,Y 431.663,Z 968.387,A -85,B 0,C 180,E1 19968.913,E2 19968.913} C_VEL
LIN {X 0,Y 428.435,Z 956.828,A -85,B 0,C 180,E1 19979.044,E2 19979.044} C_VEL
LIN {X 0,Y 431.434,Z 966.672,A -85,B 0,C 180,E1 19989.164,E2 19989.164} C_VEL
LIN {X 0,Y 440.195,Z 986.913,A -85,B 0,C 180,E1 19997.633,E2 19997.633} C_VEL
LIN {X 0,Y 450.655,Z 1019.005,A -85,B 0,C 180,E1 20005.459,E2 20005.459} C_VEL
LIN {X 0,Y 451.468,Z 1028.759,A -85,B 0,C 180,E1 20006.99,E2 20006.99} C_VEL
LIN {X 0,Y 424.197,Z 1096.613,A -85,B 0,C 180,E1 20011.596,E2 20011.596} C_VEL
LIN {X 0,Y 392.972,Z 1158.127,A -85,B 0,C 180,E1 20018.53,E2 20018.53} C_VEL
LIN {X 0,Y 363.835,Z 1209.39,A -85,B 0,C 180,E1 20028.118,E2 20028.118} C_VEL
LIN {X 0,Y 342.495,Z 1248.273,A -85,B 0,C 180,E1 20040.265,E2 20040.265} C_VEL
LIN {X 0,Y 333.163,Z 1271.443,A -85,B 0,C 180,E1 20052.772,E2 20052.772} C_VEL
LIN {X 0,Y 331.171,Z 1281.16,A -85,B 0,C 180,E1 20063.42,E2 20063.42} C_VEL
LIN {X 0,Y 331.137,Z 1282.718,A -85,B 0,C 180,E1 20071.314,E2 20071.314} C_VEL
LIN {X 0,Y 332.023,Z 1276.086,A -85,B 0,C 180,E1 20083.216,E2 20083.216} C_VEL
LIN {X 0,Y 338.485,Z 1256.742,A -85,B 0,C 180,E1 20095.964,E2 20095.964} C_VEL
LIN {X 0,Y 356.574,Z 1222.326,A -85,B 0,C 180,E1 20108.512,E2 20108.512} C_VEL
LIN {X 0,Y 384.287,Z 1173.902,A -85,B 0,C 180,E1 20119.012,E2 20119.012} C_VEL
LIN {X 0,Y 415.94,Z 1114.176,A -85,B 0,C 180,E1 20126.776,E2 20126.776} C_VEL
LIN {X 0,Y 444.922,Z 1047.499,A -85,B 0,C 180,E1 20131.953,E2 20131.953} C_VEL
LIN {X 0,Y 452.23,Z 1024.827,A -85,B 0,C 180,E1 20133.393,E2 20133.393} C_VEL
LIN {X 0,Y 451.123,Z 1020.029,A -85,B 0,C 180,E1 20134.325,E2 20134.325} C_VEL
LIN {X 0,Y 441.945,Z 1008.59,A -85,B 0,C 180,E1 20138.498,E2 20138.498} C_VEL
LIN {X 0,Y 432.038,Z 981.305,A -85,B 0,C 180,E1 20147.262,E2 20147.262} C_VEL
LIN {X 0,Y 426.685,Z 969.269,A -85,B 0,C 180,E1 20154.841,E2 20154.841} C_VEL
LIN {X 0,Y 425.874,Z 965.289,A -85,B 0,C 180,E1 20160.962,E2 20160.962} C_VEL
LIN {X 0,Y 428.408,Z 975.073,A -85,B 0,C 180,E1 20170.14,E2 20170.14} C_VEL
LIN {X 0,Y 436.069,Z 997.635,A -85,B 0,C 180,E1 20179.24,E2 20179.24} C_VEL
LIN {X 0,Y 443.486,Z 1030.218,A -85,B 0,C 180,E1 20187.06,E2 20187.06} C_VEL
LIN {X 0,Y 413.38,Z 1099.034,A -85,B 0,C 180,E1 20192.557,E2 20192.557} C_VEL
LIN {X 0,Y 380.753,Z 1157.484,A -85,B 0,C 180,E1 20200.311,E2 20200.311} C_VEL
LIN {X 0,Y 351.629,Z 1204.317,A -85,B 0,C 180,E1 20210.835,E2 20210.835} C_VEL
LIN {X 0,Y 332.523,Z 1236.576,A -85,B 0,C 180,E1 20223.255,E2 20223.255} C_VEL
LIN {X 0,Y 324.298,Z 1255.167,A -85,B 0,C 180,E1 20236.463,E2 20236.463} C_VEL
LIN {X 0,Y 323.01,Z 1261.259,A -85,B 0,C 180,E1 20248.653,E2 20248.653} C_VEL
LIN {X 0,Y 323.643,Z 1258.249,A -85,B 0,C 180,E1 20259.449,E2 20259.449} C_VEL
LIN {X 0,Y 328.653,Z 1244.06,A -85,B 0,C 180,E1 20272.4,E2 20272.4} C_VEL
LIN {X 0,Y 344.825,Z 1215.137,A -85,B 0,C 180,E1 20285.638,E2 20285.638} C_VEL
LIN {X 0,Y 371.767,Z 1172.088,A -85,B 0,C 180,E1 20296.879,E2 20296.879} C_VEL
LIN {X 0,Y 403.834,Z 1117.099,A -85,B 0,C 180,E1 20305.354,E2 20305.354} C_VEL
LIN {X 0,Y 434.562,Z 1053.385,A -85,B 0,C 180,E1 20311.212,E2 20311.212} C_VEL
LIN {X 0,Y 443.282,Z 1029.709,A -85,B 0,C 180,E1 20312.947,E2 20312.947} C_VEL
LIN {X 0,Y 435.348,Z 995.643,A -85,B 0,C 180,E1 20321.255,E2 20321.255} C_VEL
LIN {X 0,Y 428.296,Z 974.483,A -85,B 0,C 180,E1 20329.857,E2 20329.857} C_VEL
LIN {X 0,Y 425.85,Z 964.505,A -85,B 0,C 180,E1 20339.038,E2 20339.038} C_VEL
LIN {X 0,Y 428.856,Z 974.4,A -85,B 0,C 180,E1 20349.219,E2 20349.219} C_VEL
LIN {X 0,Y 437.84,Z 996.691,A -85,B 0,C 180,E1 20358.274,E2 20358.274} C_VEL
LIN {X 0,Y 447.137,Z 1029.81,A -85,B 0,C 180,E1 20366.073,E2 20366.073} C_VEL
LIN {X 0,Y 418.162,Z 1099.975,A -85,B 0,C 180,E1 20370.951,E2 20370.951} C_VEL
LIN {X 0,Y 386.149,Z 1160.723,A -85,B 0,C 180,E1 20377.984,E2 20377.984} C_VEL
LIN {X 0,Y 356.075,Z 1211.568,A -85,B 0,C 180,E1 20387.818,E2 20387.818} C_VEL
LIN {X 0,Y 334.38,Z 1249.649,A -85,B 0,C 180,E1 20400.255,E2 20400.255} C_VEL
LIN {X 0,Y 324.942,Z 1272.469,A -85,B 0,C 180,E1 20413.437,E2 20413.437} C_VEL
LIN {X 0,Y 323.168,Z 1280.895,A -85,B 0,C 180,E1 20423.256,E2 20423.256} C_VEL
LIN {X 0,Y 323.134,Z 1282.455,A -85,B 0,C 180,E1 20431.347,E2 20431.347} C_VEL
LIN {X 0,Y 324.077,Z 1275.818,A -85,B 0,C 180,E1 20443.547,E2 20443.547} C_VEL
LIN {X 0,Y 331.21,Z 1256.102,A -85,B 0,C 180,E1 20456.775,E2 20456.775} C_VEL
LIN {X 0,Y 351.173,Z 1220.055,A -85,B 0,C 180,E1 20469.938,E2 20469.938} C_VEL
LIN {X 0,Y 380.35,Z 1170.988,A -85,B 0,C 180,E1 20480.42,E2 20480.42} C_VEL
LIN {X 0,Y 412.144,Z 1112.558,A -85,B 0,C 180,E1 20487.876,E2 20487.876} C_VEL
LIN {X 0,Y 441.431,Z 1046.365,A -85,B 0,C 180,E1 20492.952,E2 20492.952} C_VEL
LIN {X 0,Y 447.08,Z 1028.675,A -85,B 0,C 180,E1 20494.139,E2 20494.139} C_VEL
LIN {X 0,Y 441.945,Z 1008.59,A -85,B 0,C 180,E1 20498.498,E2 20498.498} C_VEL
LIN {X 0,Y 433.3,Z 1000.715,A -85,B 0,C 180,E1 20502.915,E2 20502.915} C_VEL
LIN {X 0,Y 425.661,Z 980.616,A -85,B 0,C 180,E1 20511.744,E2 20511.744} C_VEL
LIN {X 0,Y 423.294,Z 972.924,A -85,B 0,C 180,E1 20520.968,E2 20520.968} C_VEL
LIN {X 0,Y 425.464,Z 982.757,A -85,B 0,C 180,E1 20530.211,E2 20530.211} C_VEL
LIN {X 0,Y 432.187,Z 1004.078,A -85,B 0,C 180,E1 20538.888,E2 20538.888} C_VEL
LIN {X 0,Y 438.432,Z 1034.497,A -85,B 0,C 180,E1 20546.408,E2 20546.408} C_VEL
LIN {X 0,Y 408.442,Z 1100.411,A -85,B 0,C 180,E1 20551.703,E2 20551.703} C_VEL
LIN {X 0,Y 375.443,Z 1157.748,A -85,B 0,C 180,E1 20559.345,E2 20559.345} C_VEL
LIN {X 0,Y 345.226,Z 1204.611,A -85,B 0,C 180,E1 20569.974,E2 20569.974} C_VEL
LIN {X 0,Y 325.06,Z 1237.046,A -85,B 0,C 180,E1 20582.706,E2 20582.706} C_VEL
LIN {X 0,Y 316.397,Z 1255.433,A -85,B 0,C 180,E1 20596.118,E2 20596.118} C_VEL
LIN {X 0,Y 315.013,Z 1261.521,A -85,B 0,C 180,E1 20608.618,E2 20608.618} C_VEL
LIN {X 0,Y 315.755,Z 1258.106,A -85,B 0,C 180,E1 20620.38,E2 20620.38} C_VEL
LIN {X 0,Y 321.678,Z 1243.213,A -85,B 0,C 180,E1 20633.649,E2 20633.649} C_VEL
LIN {X 0,Y 339.503,Z 1213.382,A -85,B 0,C 180,E1 20647.132,E2 20647.132} C_VEL
LIN {X 0,Y 367.99,Z 1169.488,A -85,B 0,C 180,E1 20658.393,E2 20658.393} C_VEL
LIN {X 0,Y 400.932,Z 1114.307,A -85,B 0,C 180,E1 20666.68,E2 20666.68} C_VEL
LIN {X 0,Y 432.408,Z 1049.694,A -85,B 0,C 180,E1 20672.433,E2 20672.433} C_VEL
LIN {X 0,Y 438.149,Z 1033.34,A -85,B 0,C 180,E1 20673.733,E2 20673.733} C_VEL
LIN {X 0,Y 431.037,Z 1000.488,A -85,B 0,C 180,E1 20682.123,E2 20682.123} C_VEL
LIN {X 0,Y 424.597,Z 979.413,A -85,B 0,C 180,E1 20691.417,E2 20691.417} C_VEL
LIN {X 0,Y 423.251,Z 972.196,A -85,B 0,C 180,E1 20699.032,E2 20699.032} C_VEL
LIN {X 0,Y 426.578,Z 983.054,A -85,B 0,C 180,E1 20709.901,E2 20709.901} C_VEL
LIN {X 0,Y 435.069,Z 1006.438,A -85,B 0,C 180,E1 20718.879,E2 20718.879} C_VEL
LIN {X 0,Y 441.759,Z 1035.15,A -85,B 0,C 180,E1 20725.458,E2 20725.458} C_VEL
LIN {X 0,Y 411.893,Z 1104.023,A -85,B 0,C 180,E1 20730.358,E2 20730.358} C_VEL
LIN {X 0,Y 378.96,Z 1164.034,A -85,B 0,C 180,E1 20737.528,E2 20737.528} C_VEL
LIN {X 0,Y 348.346,Z 1213.747,A -85,B 0,C 180,E1 20747.508,E2 20747.508} C_VEL
LIN {X 0,Y 326.692,Z 1250.189,A -85,B 0,C 180,E1 20759.88,E2 20759.88} C_VEL
LIN {X 0,Y 317.059,Z 1272.198,A -85,B 0,C 180,E1 20773.013,E2 20773.013} C_VEL
LIN {X 0,Y 315.166,Z 1280.63,A -85,B 0,C 180,E1 20783.084,E2 20783.084} C_VEL
LIN {X 0,Y 315.13,Z 1282.193,A -85,B 0,C 180,E1 20791.381,E2 20791.381} C_VEL
LIN {X 0,Y 316.13,Z 1275.55,A -85,B 0,C 180,E1 20803.894,E2 20803.894} C_VEL
LIN {X 0,Y 323.41,Z 1256.554,A -85,B 0,C 180,E1 20817.076,E2 20817.076} C_VEL
LIN {X 0,Y 342.836,Z 1222.886,A -85,B 0,C 180,E1 20829.948,E2 20829.948} C_VEL
LIN {X 0,Y 372.31,Z 1175.238,A -85,B 0,C 180,E1 20840.645,E2 20840.645} C_VEL
LIN {X 0,Y 405.776,Z 1116.145,A -85,B 0,C 180,E1 20848.481,E2 20848.481} C_VEL
LIN {X 0,Y 435.679,Z 1051.524,A -85,B 0,C 180,E1 20853.577,E2 20853.577} C_VEL
LIN {X 0,Y 442.051,Z 1032.708,A -85,B 0,C 180,E1 20854.862,E2 20854.862} C_VEL
LIN {X 0,Y 433.59,Z 1001.57,A -85,B 0,C 180,E1 20862.637,E2 20862.637} C_VEL
LIN {X 0,Y 433.3,Z 1000.715,A -85,B 0,C 180,E1 20862.915,E2 20862.915} C_VEL
LIN {X 0,Y 425.692,Z 996.019,A -85,B 0,C 180,E1 20867.522,E2 20867.522} C_VEL
LIN {X 0,Y 421.254,Z 984.378,A -85,B 0,C 180,E1 20874.775,E2 20874.775} C_VEL
LIN {X 0,Y 420.521,Z 980.471,A -85,B 0,C 180,E1 20880.974,E2 20880.974} C_VEL
LIN {X 0,Y 422.518,Z 990.447,A -85,B 0,C 180,E1 20890.283,E2 20890.283} C_VEL
LIN {X 0,Y 428.671,Z 1012.508,A -85,B 0,C 180,E1 20899.129,E2 20899.129} C_VEL
LIN {X 0,Y 433.013,Z 1040.142,A -85,B 0,C 180,E1 20905.859,E2 20905.859} C_VEL
LIN {X 0,Y 402.128,Z 1104.548,A -85,B 0,C 180,E1 20911.115,E2 20911.115} C_VEL
LIN {X 0,Y 368.2,Z 1161.178,A -85,B 0,C 180,E1 20918.9,E2 20918.9} C_VEL
LIN {X 0,Y 337.605,Z 1206.79,A -85,B 0,C 180,E1 20929.639,E2 20929.639} C_VEL
LIN {X 0,Y 316.74,Z 1238.977,A -85,B 0,C 180,E1 20942.913,E2 20942.913} C_VEL
LIN {X 0,Y 308.521,Z 1255.699,A -85,B 0,C 180,E1 20955.756,E2 20955.756} C_VEL
LIN {X 0,Y 307.016,Z 1261.784,A -85,B 0,C 180,E1 20968.582,E2 20968.582} C_VEL
LIN {X 0,Y 307.703,Z 1258.78,A -85,B 0,C 180,E1 20979.943,E2 20979.943} C_VEL
LIN {X 0,Y 313.505,Z 1244.698,A -85,B 0,C 180,E1 20993.48,E2 20993.48} C_VEL
LIN {X 0,Y 331.268,Z 1216.052,A -85,B 0,C 180,E1 21007.179,E2 21007.179} C_VEL
LIN {X 0,Y 360.188,Z 1173.282,A -85,B 0,C 180,E1 21018.679,E2 21018.679} C_VEL
LIN {X 0,Y 394.433,Z 1118.132,A -85,B 0,C 180,E1 21027.264,E2 21027.264} C_VEL
LIN {X 0,Y 426.694,Z 1054.539,A -85,B 0,C 180,E1 21033.085,E2 21033.085} C_VEL
LIN {X 0,Y 433.166,Z 1037.947,A -85,B 0,C 180,E1 21034.346,E2 21034.346} C_VEL
LIN {X 0,Y 427.216,Z 1006.948,A -85,B 0,C 180,E1 21042.492,E2 21042.492} C_VEL
LIN {X 0,Y 421.411,Z 985.689,A -85,B 0,C 180,E1 21052.165,E2 21052.165} C_VEL
LIN {X 0,Y 420.489,Z 979.811,A -85,B 0,C 180,E1 21059.026,E2 21059.026} C_VEL
LIN {X 0,Y 423.339,Z 990.006,A -85,B 0,C 180,E1 21069.545,E2 21069.545} C_VEL
LIN {X 0,Y 431.117,Z 1012.843,A -85,B 0,C 180,E1 21078.526,E2 21078.526} C_VEL
LIN {X 0,Y 436.682,Z 1039.13,A -85,B 0,C 180,E1 21084.709,E2 21084.709} C_VEL
LIN {X 0,Y 405.509,Z 1108.218,A -85,B 0,C 180,E1 21089.767,E2 21089.767} C_VEL
LIN {X 0,Y 371.411,Z 1167.874,A -85,B 0,C 180,E1 21097.152,E2 21097.152} C_VEL
LIN {X 0,Y 339.584,Z 1217.375,A -85,B 0,C 180,E1 21107.601,E2 21107.601} C_VEL
LIN {X 0,Y 317.645,Z 1253.2,A -85,B 0,C 180,E1 21120.668,E2 21120.668} C_VEL
LIN {X 0,Y 308.644,Z 1273.885,A -85,B 0,C 180,E1 21134.305,E2 21134.305} C_VEL
LIN {X 0,Y 307.125,Z 1281.447,A -85,B 0,C 180,E1 21145.749,E2 21145.749} C_VEL
LIN {X 0,Y 307.193,Z 1280.37,A -85,B 0,C 180,E1 21157.098,E2 21157.098} C_VEL
LIN {X 0,Y 310.865,Z 1267.755,A -85,B 0,C 180,E1 21170.736,E2 21170.736} C_VEL
LIN {X 0,Y 324.755,Z 1240.991,A -85,B 0,C 180,E1 21184.639,E2 21184.639} C_VEL
LIN {X 0,Y 351.225,Z 1199.546,A -85,B 0,C 180,E1 21196.837,E2 21196.837} C_VEL
LIN {X 0,Y 384.95,Z 1145.412,A -85,B 0,C 180,E1 21206.102,E2 21206.102} C_VEL
LIN {X 0,Y 418.945,Z 1080.763,A -85,B 0,C 180,E1 21212.599,E2 21212.599} C_VEL
LIN {X 0,Y 437.122,Z 1036.986,A -85,B 0,C 180,E1 21215.557,E2 21215.557} C_VEL
LIN {X 0,Y 429.493,Z 1007.399,A -85,B 0,C 180,E1 21223.207,E2 21223.207} C_VEL
LIN {X 0,Y 425.692,Z 996.019,A -85,B 0,C 180,E1 21227.522,E2 21227.522} C_VEL
LIN {X 0,Y 419.484,Z 994.766,A -85,B 0,C 180,E1 21232.28,E2 21232.28} C_VEL
LIN {X 0,Y 417.564,Z 988.081,A -85,B 0,C 180,E1 21241.104,E2 21241.104} C_VEL
LIN {X 0,Y 419.319,Z 998.08,A -85,B 0,C 180,E1 21250.362,E2 21250.362} C_VEL
LIN {X 0,Y 424.755,Z 1020.116,A -85,B 0,C 180,E1 21259.157,E2 21259.157} C_VEL
LIN {X 0,Y 427.688,Z 1044.824,A -85,B 0,C 180,E1 21265.156,E2 21265.156} C_VEL
LIN {X 0,Y 395.333,Z 1109.617,A -85,B 0,C 180,E1 21270.607,E2 21270.607} C_VEL
LIN {X 0,Y 359.967,Z 1166.084,A -85,B 0,C 180,E1 21278.719,E2 21278.719} C_VEL
LIN {X 0,Y 329.071,Z 1210.095,A -85,B 0,C 180,E1 21289.648,E2 21289.648} C_VEL
LIN {X 0,Y 307.859,Z 1241.681,A -85,B 0,C 180,E1 21303.652,E2 21303.652} C_VEL
LIN {X 0,Y 300.23,Z 1257.131,A -85,B 0,C 180,E1 21316.847,E2 21316.847} C_VEL
LIN {X 0,Y 299.018,Z 1262.046,A -85,B 0,C 180,E1 21328.545,E2 21328.545} C_VEL
LIN {X 0,Y 299.746,Z 1259.046,A -85,B 0,C 180,E1 21340.21,E2 21340.21} C_VEL
LIN {X 0,Y 305.93,Z 1245.058,A -85,B 0,C 180,E1 21354.035,E2 21354.035} C_VEL
LIN {X 0,Y 324.935,Z 1216.013,A -85,B 0,C 180,E1 21368.17,E2 21368.17} C_VEL
LIN {X 0,Y 355.25,Z 1172.858,A -85,B 0,C 180,E1 21379.823,E2 21379.823} C_VEL
LIN {X 0,Y 390.148,Z 1118.271,A -85,B 0,C 180,E1 21388.29,E2 21388.29} C_VEL
LIN {X 0,Y 423.188,Z 1054.545,A -85,B 0,C 180,E1 21394.087,E2 21394.087} C_VEL
LIN {X 0,Y 428.166,Z 1041.964,A -85,B 0,C 180,E1 21395.102,E2 21395.102} C_VEL
LIN {X 0,Y 422.897,Z 1011.907,A -85,B 0,C 180,E1 21403.383,E2 21403.383} C_VEL
LIN {X 0,Y 418.223,Z 992.488,A -85,B 0,C 180,E1 21412.766,E2 21412.766} C_VEL
LIN {X 0,Y 417.518,Z 987.998,A -85,B 0,C 180,E1 21421.101,E2 21421.101} C_VEL
LIN {X 0,Y 421.226,Z 1000.147,A -85,B 0,C 180,E1 21430.96,E2 21430.96} C_VEL
LIN {X 0,Y 428.422,Z 1024.73,A -85,B 0,C 180,E1 21439.721,E2 21439.721} C_VEL
LIN {X 0,Y 431.386,Z 1043.491,A -85,B 0,C 180,E1 21443.982,E2 21443.982} C_VEL
LIN {X 0,Y 399.539,Z 1111.439,A -85,B 0,C 180,E1 21449.083,E2 21449.083} C_VEL
LIN {X 0,Y 364.649,Z 1170.27,A -85,B 0,C 180,E1 21456.556,E2 21456.556} C_VEL
LIN {X 0,Y 332.182,Z 1218.832,A -85,B 0,C 180,E1 21467.126,E2 21467.126} C_VEL
LIN {X 0,Y 309.538,Z 1254.304,A -85,B 0,C 180,E1 21480.631,E2 21480.631} C_VEL
LIN {X 0,Y 300.762,Z 1273.615,A -85,B 0,C 180,E1 21493.883,E2 21493.883} C_VEL
LIN {X 0,Y 299.115,Z 1281.183,A -85,B 0,C 180,E1 21505.635,E2 21505.635} C_VEL
LIN {X 0,Y 299.193,Z 1280.106,A -85,B 0,C 180,E1 21517.289,E2 21517.289} C_VEL
LIN {X 0,Y 303.121,Z 1267.484,A -85,B 0,C 180,E1 21531.292,E2 21531.292} C_VEL
LIN {X 0,Y 317.644,Z 1241.035,A -85,B 0,C 180,E1 21545.379,E2 21545.379} C_VEL
LIN {X 0,Y 345.479,Z 1199.27,A -85,B 0,C 180,E1 21557.863,E2 21557.863} C_VEL
LIN {X 0,Y 380.516,Z 1144.88,A -85,B 0,C 180,E1 21567.18,E2 21567.18} C_VEL
LIN {X 0,Y 415.236,Z 1080.499,A -85,B 0,C 180,E1 21573.604,E2 21573.604} C_VEL
LIN {X 0,Y 432.174,Z 1041.85,A -85,B 0,C 180,E1 21576.126,E2 21576.126} C_VEL
LIN {X 0,Y 425.346,Z 1012.929,A -85,B 0,C 180,E1 21583.891,E2 21583.891} C_VEL
LIN {X 0,Y 419.484,Z 994.766,A -85,B 0,C 180,E1 21592.28,E2 21592.28} C_VEL
LIN {X 0,Y 414.644,Z 997.459,A -85,B 0,C 180,E1 21597.106,E2 21597.106} C_VEL
LIN {X 0,Y 414.277,Z 997.074,A -85,B 0,C 180,E1 21603.089,E2 21603.089} C_VEL
LIN {X 0,Y 416.524,Z 1007.583,A -85,B 0,C 180,E1 21611.496,E2 21611.496} C_VEL
LIN {X 0,Y 421.208,Z 1030.279,A -85,B 0,C 180,E1 21619.947,E2 21619.947} C_VEL
LIN {X 0,Y 422.301,Z 1049.444,A -85,B 0,C 180,E1 21624.455,E2 21624.455} C_VEL
LIN {X 0,Y 389.13,Z 1113.295,A -85,B 0,C 180,E1 21629.955,E2 21629.955} C_VEL
LIN {X 0,Y 353.661,Z 1167.95,A -85,B 0,C 180,E1 21637.984,E2 21637.984} C_VEL
LIN {X 0,Y 321.464,Z 1212.047,A -85,B 0,C 180,E1 21649.276,E2 21649.276} C_VEL
LIN {X 0,Y 299.738,Z 1243.066,A -85,B 0,C 180,E1 21663.693,E2 21663.693} C_VEL
LIN {X 0,Y 292.324,Z 1257.397,A -85,B 0,C 180,E1 21676.484,E2 21676.484} C_VEL
LIN {X 0,Y 291.028,Z 1262.308,A -85,B 0,C 180,E1 21688.505,E2 21688.505} C_VEL
LIN {X 0,Y 291.784,Z 1259.312,A -85,B 0,C 180,E1 21700.491,E2 21700.491} C_VEL
LIN {X 0,Y 298.528,Z 1245.154,A -85,B 0,C 180,E1 21714.797,E2 21714.797} C_VEL
LIN {X 0,Y 318.718,Z 1215.94,A -85,B 0,C 180,E1 21729.213,E2 21729.213} C_VEL
LIN {X 0,Y 350.179,Z 1172.796,A -85,B 0,C 180,E1 21740.932,E2 21740.932} C_VEL
LIN {X 0,Y 385.884,Z 1118.545,A -85,B 0,C 180,E1 21749.33,E2 21749.33} C_VEL
LIN {X 0,Y 419.679,Z 1054.861,A -85,B 0,C 180,E1 21755.082,E2 21755.082} C_VEL
LIN {X 0,Y 423.075,Z 1045.387,A -85,B 0,C 180,E1 21756.018,E2 21756.018} C_VEL
LIN {X 0,Y 418.551,Z 1016.837,A -85,B 0,C 180,E1 21764.287,E2 21764.287} C_VEL
LIN {X 0,Y 414.999,Z 999.968,A -85,B 0,C 180,E1 21772.709,E2 21772.709} C_VEL
LIN {X 0,Y 414.587,Z 995.511,A -85,B 0,C 180,E1 21781.109,E2 21781.109} C_VEL
LIN {X 0,Y 417.928,Z 1007.745,A -85,B 0,C 180,E1 21791.048,E2 21791.048} C_VEL
LIN {X 0,Y 424.148,Z 1031.01,A -85,B 0,C 180,E1 21799.384,E2 21799.384} C_VEL
LIN {X 0,Y 426.339,Z 1047.435,A -85,B 0,C 180,E1 21803.215,E2 21803.215} C_VEL
LIN {X 0,Y 392.976,Z 1115.834,A -85,B 0,C 180,E1 21808.496,E2 21808.496} C_VEL
LIN {X 0,Y 356.655,Z 1174.556,A -85,B 0,C 180,E1 21816.257,E2 21816.257} C_VEL
LIN {X 0,Y 323.611,Z 1222.004,A -85,B 0,C 180,E1 21827.14,E2 21827.14} C_VEL
LIN {X 0,Y 301.441,Z 1255.409,A -85,B 0,C 180,E1 21840.593,E2 21840.593} C_VEL
LIN {X 0,Y 292.444,Z 1274.872,A -85,B 0,C 180,E1 21855.118,E2 21855.118} C_VEL
LIN {X 0,Y 291.45,Z 1281.414,A -85,B 0,C 180,E1 21868.508,E2 21868.508} C_VEL
LIN {X 0,Y 291.8,Z 1277.262,A -85,B 0,C 180,E1 21882.012,E2 21882.012} C_VEL
LIN {X 0,Y 298.563,Z 1260.476,A -85,B 0,C 180,E1 21896.502,E2 21896.502} C_VEL
LIN {X 0,Y 319.371,Z 1228.387,A -85,B 0,C 180,E1 21910.815,E2 21910.815} C_VEL
LIN {X 0,Y 350.809,Z 1183.33,A -85,B 0,C 180,E1 21922.165,E2 21922.165} C_VEL
LIN {X 0,Y 386.45,Z 1127.332,A -85,B 0,C 180,E1 21930.322,E2 21930.322} C_VEL
LIN {X 0,Y 419.662,Z 1063.443,A -85,B 0,C 180,E1 21935.765,E2 21935.765} C_VEL
LIN {X 0,Y 427.121,Z 1045.804,A -85,B 0,C 180,E1 21936.898,E2 21936.898} C_VEL
LIN {X 0,Y 421.437,Z 1019.336,A -85,B 0,C 180,E1 21944.274,E2 21944.274} C_VEL
LIN {X 0,Y 416.159,Z 1001.701,A -85,B 0,C 180,E1 21952.609,E2 21952.609} C_VEL
LIN {X 0,Y 414.644,Z 997.459,A -85,B 0,C 180,E1 21957.106,E2 21957.106} C_VEL
LIN {X 0,Y 411.171,Z 1003.545,A -85,B 0,C 180,E1 21961.965,E2 21961.965} C_VEL
LIN {X 0,Y 412.63,Z 1013.229,A -85,B 0,C 180,E1 21970.532,E2 21970.532} C_VEL
LIN {X 0,Y 416.544,Z 1034.592,A -85,B 0,C 180,E1 21979.072,E2 21979.072} C_VEL
LIN {X 0,Y 417.222,Z 1053.509,A -85,B 0,C 180,E1 21983.693,E2 21983.693} C_VEL
LIN {X 0,Y 383.454,Z 1116.2,A -85,B 0,C 180,E1 21989.195,E2 21989.195} C_VEL
LIN {X 0,Y 345.853,Z 1171.961,A -85,B 0,C 180,E1 21997.655,E2 21997.655} C_VEL
LIN {X 0,Y 313.306,Z 1214.724,A -85,B 0,C 180,E1 22009.144,E2 22009.144} C_VEL
LIN {X 0,Y 291.599,Z 1244.452,A -85,B 0,C 180,E1 22023.734,E2 22023.734} C_VEL
LIN {X 0,Y 284.427,Z 1257.663,A -85,B 0,C 180,E1 22036.102,E2 22036.102} C_VEL
LIN {X 0,Y 283.03,Z 1262.571,A -85,B 0,C 180,E1 22048.462,E2 22048.462} C_VEL
LIN {X 0,Y 283.832,Z 1259.578,A -85,B 0,C 180,E1 22060.789,E2 22060.789} C_VEL
LIN {X 0,Y 291.828,Z 1244.297,A -85,B 0,C 180,E1 22076.242,E2 22076.242} C_VEL
LIN {X 0,Y 313.615,Z 1214.482,A -85,B 0,C 180,E1 22090.805,E2 22090.805} C_VEL
LIN {X 0,Y 346.732,Z 1170.779,A -85,B 0,C 180,E1 22102.45,E2 22102.45} C_VEL
LIN {X 0,Y 383.922,Z 1115.263,A -85,B 0,C 180,E1 22110.805,E2 22110.805} C_VEL
LIN {X 0,Y 418.088,Z 1050.084,A -85,B 0,C 180,E1 22116.628,E2 22116.628} C_VEL
LIN {X 0,Y 414.486,Z 1022.958,A -85,B 0,C 180,E1 22124.775,E2 22124.775} C_VEL
LIN {X 0,Y 411.705,Z 1007.476,A -85,B 0,C 180,E1 22132.651,E2 22132.651} C_VEL
LIN {X 0,Y 411.335,Z 1002.889,A -85,B 0,C 180,E1 22141.117,E2 22141.117} C_VEL
LIN {X 0,Y 414.614,Z 1015.331,A -85,B 0,C 180,E1 22151.123,E2 22151.123} C_VEL
LIN {X 0,Y 420.192,Z 1039.16,A -85,B 0,C 180,E1 22159.574,E2 22159.574} C_VEL
LIN {X 0,Y 421.019,Z 1052.234,A -85,B 0,C 180,E1 22162.482,E2 22162.482} C_VEL
LIN {X 0,Y 386.433,Z 1120.227,A -85,B 0,C 180,E1 22167.882,E2 22167.882} C_VEL
LIN {X 0,Y 348.917,Z 1178.443,A -85,B 0,C 180,E1 22175.87,E2 22175.87} C_VEL
LIN {X 0,Y 315.097,Z 1225.051,A -85,B 0,C 180,E1 22187.116,E2 22187.116} C_VEL
LIN {X 0,Y 292.64,Z 1257.723,A -85,B 0,C 180,E1 22201.22,E2 22201.22} C_VEL
LIN {X 0,Y 284.169,Z 1275.734,A -85,B 0,C 180,E1 22216.091,E2 22216.091} C_VEL
LIN {X 0,Y 283.435,Z 1281.151,A -85,B 0,C 180,E1 22228.466,E2 22228.466} C_VEL
LIN {X 0,Y 283.856,Z 1276.995,A -85,B 0,C 180,E1 22242.354,E2 22242.354} C_VEL
LIN {X 0,Y 291.147,Z 1260.204,A -85,B 0,C 180,E1 22257.232,E2 22257.232} C_VEL
LIN {X 0,Y 313.061,Z 1228.113,A -85,B 0,C 180,E1 22271.82,E2 22271.82} C_VEL
LIN {X 0,Y 346.477,Z 1181.999,A -85,B 0,C 180,E1 22283.47,E2 22283.47} C_VEL
LIN {X 0,Y 383.565,Z 1125.162,A -85,B 0,C 180,E1 22291.615,E2 22291.615} C_VEL
LIN {X 0,Y 417.619,Z 1060.496,A -85,B 0,C 180,E1 22296.963,E2 22296.963} C_VEL
LIN {X 0,Y 421.947,Z 1048.683,A -85,B 0,C 180,E1 22297.958,E2 22297.958} C_VEL
LIN {X 0,Y 416.62,Z 1022.866,A -85,B 0,C 180,E1 22305.708,E2 22305.708} C_VEL
LIN {X 0,Y 412.055,Z 1006.723,A -85,B 0,C 180,E1 22314.658,E2 22314.658} C_VEL
LIN {X 0,Y 411.171,Z 1003.545,A -85,B 0,C 180,E1 22321.965,E2 22321.965} C_VEL
LIN {X 0,Y 408.138,Z 1014.72,A -85,B 0,C 180,E1 22326.66,E2 22326.66} C_VEL
LIN {X 0,Y 411.06,Z 1032.722,A -85,B 0,C 180,E1 22336.007,E2 22336.007} C_VEL
LIN {X 0,Y 412.593,Z 1056.783,A -85,B 0,C 180,E1 22342.861,E2 22342.861} C_VEL
LIN {X 0,Y 377.469,Z 1119.718,A -85,B 0,C 180,E1 22348.483,E2 22348.483} C_VEL
LIN {X 0,Y 338.78,Z 1174.983,A -85,B 0,C 180,E1 22357.106,E2 22357.106} C_VEL
LIN {X 0,Y 305.535,Z 1216.906,A -85,B 0,C 180,E1 22368.824,E2 22368.824} C_VEL
LIN {X 0,Y 283.465,Z 1245.837,A -85,B 0,C 180,E1 22383.778,E2 22383.778} C_VEL
LIN {X 0,Y 275.784,Z 1259.904,A -85,B 0,C 180,E1 22398.891,E2 22398.891} C_VEL
LIN {X 0,Y 275.293,Z 1262.814,A -85,B 0,C 180,E1 22411.579,E2 22411.579} C_VEL
LIN {X 0,Y 277.213,Z 1256.683,A -85,B 0,C 180,E1 22425.891,E2 22425.891} C_VEL
LIN {X 0,Y 289.446,Z 1237.291,A -85,B 0,C 180,E1 22441.633,E2 22441.633} C_VEL
LIN {X 0,Y 315.911,Z 1203.883,A -85,B 0,C 180,E1 22455.492,E2 22455.492} C_VEL
LIN {X 0,Y 352.248,Z 1156.798,A -85,B 0,C 180,E1 22466.181,E2 22466.181} C_VEL
LIN {X 0,Y 390.14,Z 1098.614,A -85,B 0,C 180,E1 22473.667,E2 22473.667} C_VEL
LIN {X 0,Y 413.139,Z 1054.229,A -85,B 0,C 180,E1 22477.385,E2 22477.385} C_VEL
LIN {X 0,Y 410.294,Z 1028.252,A -85,B 0,C 180,E1 22485.609,E2 22485.609} C_VEL
LIN {X 0,Y 408.286,Z 1014.927,A -85,B 0,C 180,E1 22492.589,E2 22492.589} C_VEL
LIN {X 0,Y 408.084,Z 1010.239,A -85,B 0,C 180,E1 22501.126,E2 22501.126} C_VEL
LIN {X 0,Y 410.731,Z 1021.773,A -85,B 0,C 180,E1 22510.676,E2 22510.676} C_VEL
LIN {X 0,Y 415.652,Z 1045.291,A -85,B 0,C 180,E1 22519.242,E2 22519.242} C_VEL
LIN {X 0,Y 415.849,Z 1056.654,A -85,B 0,C 180,E1 22521.719,E2 22521.719} C_VEL
LIN {X 0,Y 379.917,Z 1124.384,A -85,B 0,C 180,E1 22527.25,E2 22527.25} C_VEL
LIN {X 0,Y 342.112,Z 1180.79,A -85,B 0,C 180,E1 22535.224,E2 22535.224} C_VEL
LIN {X 0,Y 308.117,Z 1225.826,A -85,B 0,C 180,E1 22546.409,E2 22546.409} C_VEL
LIN {X 0,Y 284.732,Z 1258.412,A -85,B 0,C 180,E1 22561.014,E2 22561.014} C_VEL
LIN {X 0,Y 276.256,Z 1275.466,A -85,B 0,C 180,E1 22575.684,E2 22575.684} C_VEL
LIN {X 0,Y 275.419,Z 1280.887,A -85,B 0,C 180,E1 22588.422,E2 22588.422} C_VEL
LIN {X 0,Y 275.643,Z 1277.64,A -85,B 0,C 180,E1 22601.115,E2 22601.115} C_VEL
LIN {X 0,Y 282.246,Z 1262.427,A -85,B 0,C 180,E1 22616.344,E2 22616.344} C_VEL
LIN {X 0,Y 302.599,Z 1233.325,A -85,B 0,C 180,E1 22630.949,E2 22630.949} C_VEL
LIN {X 0,Y 336.254,Z 1188.944,A -85,B 0,C 180,E1 22643.185,E2 22643.185} C_VEL
LIN {X 0,Y 374.33,Z 1133.563,A -85,B 0,C 180,E1 22651.745,E2 22651.745} C_VEL
LIN {X 0,Y 409.953,Z 1069.772,A -85,B 0,C 180,E1 22657.404,E2 22657.404} C_VEL
LIN {X 0,Y 417.116,Z 1053.411,A -85,B 0,C 180,E1 22658.605,E2 22658.605} C_VEL
LIN {X 0,Y 412.588,Z 1029.183,A -85,B 0,C 180,E1 22666.109,E2 22666.109} C_VEL
LIN {X 0,Y 408.805,Z 1014.102,A -85,B 0,C 180,E1 22674.615,E2 22674.615} C_VEL
LIN {X 0,Y 407.945,Z 1010.8,A -85,B 0,C 180,E1 22681.846,E2 22681.846} C_VEL
LIN {X 0,Y 408.138,Z 1014.72,A -85,B 0,C 180,E1 22686.66,E2 22686.66} C_VEL
LIN {X 0,Y 405.502,Z 1029.083,A -85,B 0,C 180,E1 22691.242,E2 22691.242} C_VEL
LIN {X 0,Y 407.928,Z 1051.627,A -85,B 0,C 180,E1 22699.806,E2 22699.806} C_VEL
LIN {X 0,Y 407.006,Z 1062.24,A -85,B 0,C 180,E1 22702.16,E2 22702.16} C_VEL
LIN {X 0,Y 370.562,Z 1124.84,A -85,B 0,C 180,E1 22707.947,E2 22707.947} C_VEL
LIN {X 0,Y 331.236,Z 1178.638,A -85,B 0,C 180,E1 22716.672,E2 22716.672} C_VEL
LIN {X 0,Y 296.204,Z 1220.831,A -85,B 0,C 180,E1 22729.195,E2 22729.195} C_VEL
LIN {X 0,Y 275.367,Z 1247.221,A -85,B 0,C 180,E1 22743.828,E2 22743.828} C_VEL
LIN {X 0,Y 267.837,Z 1260.169,A -85,B 0,C 180,E1 22758.557,E2 22758.557} C_VEL
LIN {X 0,Y 267.287,Z 1263.077,A -85,B 0,C 180,E1 22771.626,E2 22771.626} C_VEL
LIN {X 0,Y 269.331,Z 1257.052,A -85,B 0,C 180,E1 22786.223,E2 22786.223} C_VEL
LIN {X 0,Y 282.375,Z 1237.566,A -85,B 0,C 180,E1 22802.521,E2 22802.521} C_VEL
LIN {X 0,Y 309.816,Z 1204.512,A -85,B 0,C 180,E1 22816.482,E2 22816.482} C_VEL
LIN {X 0,Y 347.18,Z 1157.767,A -85,B 0,C 180,E1 22827.195,E2 22827.195} C_VEL
LIN {X 0,Y 385.612,Z 1100.467,A -85,B 0,C 180,E1 22834.602,E2 22834.602} C_VEL
LIN {X 0,Y 408.195,Z 1058.666,A -85,B 0,C 180,E1 22838.114,E2 22838.114} C_VEL
LIN {X 0,Y 406.096,Z 1034.499,A -85,B 0,C 180,E1 22846.009,E2 22846.009} C_VEL
LIN {X 0,Y 404.19,Z 1020.315,A -85,B 0,C 180,E1 22854.677,E2 22854.677} C_VEL
LIN {X 0,Y 404.671,Z 1017.535,A -85,B 0,C 180,E1 22861.136,E2 22861.136} C_VEL
LIN {X 0,Y 407.068,Z 1029.264,A -85,B 0,C 180,E1 22870.773,E2 22870.773} C_VEL
LIN {X 0,Y 411.133,Z 1051.414,A -85,B 0,C 180,E1 22878.903,E2 22878.903} C_VEL
LIN {X 0,Y 411.075,Z 1060.112,A -85,B 0,C 180,E1 22880.893,E2 22880.893} C_VEL
LIN {X 0,Y 374.454,Z 1126.816,A -85,B 0,C 180,E1 22886.42,E2 22886.42} C_VEL
LIN {X 0,Y 334.744,Z 1183.827,A -85,B 0,C 180,E1 22894.691,E2 22894.691} C_VEL
LIN {X 0,Y 298.85,Z 1229.503,A -85,B 0,C 180,E1 22906.704,E2 22906.704} C_VEL
LIN {X 0,Y 275.647,Z 1260.943,A -85,B 0,C 180,E1 22922.088,E2 22922.088} C_VEL
LIN {X 0,Y 267.992,Z 1276.451,A -85,B 0,C 180,E1 22936.905,E2 22936.905} C_VEL
LIN {X 0,Y 267.404,Z 1280.624,A -85,B 0,C 180,E1 22948.374,E2 22948.374} C_VEL
LIN {X 0,Y 267.677,Z 1277.374,A -85,B 0,C 180,E1 22961.45,E2 22961.45} C_VEL
LIN {X 0,Y 274.808,Z 1262.154,A -85,B 0,C 180,E1 22977.114,E2 22977.114} C_VEL
LIN {X 0,Y 297.16,Z 1231.994,A -85,B 0,C 180,E1 22992.388,E2 22992.388} C_VEL
LIN {X 0,Y 332.453,Z 1187.074,A -85,B 0,C 180,E1 23004.672,E2 23004.672} C_VEL
LIN {X 0,Y 372.034,Z 1130.762,A -85,B 0,C 180,E1 23013.169,E2 23013.169} C_VEL
LIN {X 0,Y 408.19,Z 1066.784,A -85,B 0,C 180,E1 23018.639,E2 23018.639} C_VEL
LIN {X 0,Y 412.092,Z 1057.315,A -85,B 0,C 180,E1 23019.463,E2 23019.463} C_VEL
LIN {X 0,Y 408.258,Z 1034.249,A -85,B 0,C 180,E1 23027.053,E2 23027.053} C_VEL
LIN {X 0,Y 405.259,Z 1021.373,A -85,B 0,C 180,E1 23034.568,E2 23034.568} C_VEL
LIN {X 0,Y 404.728,Z 1017.451,A -85,B 0,C 180,E1 23041.012,E2 23041.012} C_VEL
LIN {X 0,Y 405.465,Z 1028.8,A -85,B 0,C 180,E1 23051.093,E2 23051.093} C_VEL
LIN {X 0,Y 405.502,Z 1029.083,A -85,B 0,C 180,E1 23051.242,E2 23051.242} C_VEL
LIN {X 0,Y 402.62,Z 1046.231,A -85,B 0,C 180,E1 23055.661,E2 23055.661} C_VEL
LIN {X 0,Y 403.033,Z 1064.306,A -85,B 0,C 180,E1 23061.219,E2 23061.219} C_VEL
LIN {X 0,Y 366.11,Z 1126.098,A -85,B 0,C 180,E1 23066.933,E2 23066.933} C_VEL
LIN {X 0,Y 325.216,Z 1180.214,A -85,B 0,C 180,E1 23075.798,E2 23075.798} C_VEL
LIN {X 0,Y 289.953,Z 1221.102,A -85,B 0,C 180,E1 23088.12,E2 23088.12} C_VEL
LIN {X 0,Y 267.978,Z 1247.491,A -85,B 0,C 180,E1 23103.049,E2 23103.049} C_VEL
LIN {X 0,Y 259.893,Z 1260.435,A -85,B 0,C 180,E1 23118.202,E2 23118.202} C_VEL
LIN {X 0,Y 259.281,Z 1263.339,A -85,B 0,C 180,E1 23131.677,E2 23131.677} C_VEL
LIN {X 0,Y 261.79,Z 1256.899,A -85,B 0,C 180,E1 23147.334,E2 23147.334} C_VEL
LIN {X 0,Y 275.416,Z 1237.84,A -85,B 0,C 180,E1 23163.449,E2 23163.449} C_VEL
LIN {X 0,Y 305.001,Z 1203.819,A -85,B 0,C 180,E1 23177.924,E2 23177.924} C_VEL
LIN {X 0,Y 343.242,Z 1157.426,A -85,B 0,C 180,E1 23188.465,E2 23188.465} C_VEL
LIN {X 0,Y 383.117,Z 1099.259,A -85,B 0,C 180,E1 23195.844,E2 23195.844} C_VEL
LIN {X 0,Y 403.271,Z 1062.151,A -85,B 0,C 180,E1 23199.125,E2 23199.125} C_VEL
LIN {X 0,Y 401.68,Z 1038.289,A -85,B 0,C 180,E1 23207.495,E2 23207.495} C_VEL
LIN {X 0,Y 400.612,Z 1027.539,A -85,B 0,C 180,E1 23214.63,E2 23214.63} C_VEL
LIN {X 0,Y 401.087,Z 1024.74,A -85,B 0,C 180,E1 23221.146,E2 23221.146} C_VEL
LIN {X 0,Y 403.301,Z 1036.801,A -85,B 0,C 180,E1 23230.905,E2 23230.905} C_VEL
LIN {X 0,Y 406.713,Z 1060.095,A -85,B 0,C 180,E1 23239.321,E2 23239.321} C_VEL
LIN {X 0,Y 404.441,Z 1067.598,A -85,B 0,C 180,E1 23240.308,E2 23240.308} C_VEL
LIN {X 0,Y 366.448,Z 1133.294,A -85,B 0,C 180,E1 23246.011,E2 23246.011} C_VEL
LIN {X 0,Y 325.687,Z 1189.175,A -85,B 0,C 180,E1 23254.608,E2 23254.608} C_VEL
LIN {X 0,Y 289.617,Z 1233.23,A -85,B 0,C 180,E1 23267.047,E2 23267.047} C_VEL
LIN {X 0,Y 266.771,Z 1263.235,A -85,B 0,C 180,E1 23283.064,E2 23283.064} C_VEL
LIN {X 0,Y 259.719,Z 1277.097,A -85,B 0,C 180,E1 23298.196,E2 23298.196} C_VEL
LIN {X 0,Y 259.121,Z 1280.354,A -85,B 0,C 180,E1 23311.68,E2 23311.68} C_VEL
LIN {X 0,Y 260.535,Z 1274.551,A -85,B 0,C 180,E1 23325.735,E2 23325.735} C_VEL
LIN {X 0,Y 272.026,Z 1255.733,A -85,B 0,C 180,E1 23342.018,E2 23342.018} C_VEL
LIN {X 0,Y 300.002,Z 1220.961,A -85,B 0,C 180,E1 23357.203,E2 23357.203} C_VEL
LIN {X 0,Y 337.738,Z 1173.783,A -85,B 0,C 180,E1 23368.299,E2 23368.299} C_VEL
LIN {X 0,Y 377.896,Z 1115.488,A -85,B 0,C 180,E1 23375.884,E2 23375.884} C_VEL
LIN {X 0,Y 407.176,Z 1062.234,A -85,B 0,C 180,E1 23380.057,E2 23380.057} C_VEL
LIN {X 0,Y 403.849,Z 1039.202,A -85,B 0,C 180,E1 23388.012,E2 23388.012} C_VEL
LIN {X 0,Y 401.136,Z 1026.865,A -85,B 0,C 180,E1 23396.685,E2 23396.685} C_VEL
LIN {X 0,Y 400.684,Z 1026.217,A -85,B 0,C 180,E1 23403.194,E2 23403.194} C_VEL
LIN {X 0,Y 401.658,Z 1037.542,A -85,B 0,C 180,E1 23411.927,E2 23411.927} C_VEL
LIN {X 0,Y 402.62,Z 1046.231,A -85,B 0,C 180,E1 23415.661,E2 23415.661} C_VEL
LIN {X 0,Y 398.468,Z 1066.047,A -85,B 0,C 180,E1 23419.867,E2 23419.867} C_VEL
LIN {X 0,Y 393.149,Z 1077.374,A -85,B 0,C 180,E1 23421.048,E2 23421.048} C_VEL
LIN {X 0,Y 353.678,Z 1138.583,A -85,B 0,C 180,E1 23427.333,E2 23427.333} C_VEL
LIN {X 0,Y 312.544,Z 1189.627,A -85,B 0,C 180,E1 23436.729,E2 23436.729} C_VEL
LIN {X 0,Y 277.558,Z 1228.131,A -85,B 0,C 180,E1 23449.981,E2 23449.981} C_VEL
LIN {X 0,Y 257.873,Z 1251.396,A -85,B 0,C 180,E1 23465.54,E2 23465.54} C_VEL
LIN {X 0,Y 251.455,Z 1262.22,A -85,B 0,C 180,E1 23481.318,E2 23481.318} C_VEL
LIN {X 0,Y 251.242,Z 1263.167,A -85,B 0,C 180,E1 23495.199,E2 23495.199} C_VEL
LIN {X 0,Y 255.513,Z 1254.687,A -85,B 0,C 180,E1 23510.884,E2 23510.884} C_VEL
LIN {X 0,Y 273.481,Z 1232.493,A -85,B 0,C 180,E1 23527.633,E2 23527.633} C_VEL
LIN {X 0,Y 306.832,Z 1195.859,A -85,B 0,C 180,E1 23541.507,E2 23541.507} C_VEL
LIN {X 0,Y 348.436,Z 1145.369,A -85,B 0,C 180,E1 23551.593,E2 23551.593} C_VEL
LIN {X 0,Y 388.242,Z 1085.644,A -85,B 0,C 180,E1 23558.161,E2 23558.161} C_VEL
LIN {X 0,Y 398.304,Z 1067.089,A -85,B 0,C 180,E1 23559.709,E2 23559.709} C_VEL
LIN {X 0,Y 397.538,Z 1044.5,A -85,B 0,C 180,E1 23567.947,E2 23567.947} C_VEL
LIN {X 0,Y 396.848,Z 1034.69,A -85,B 0,C 180,E1 23574.579,E2 23574.579} C_VEL
LIN {X 0,Y 397.502,Z 1031.945,A -85,B 0,C 180,E1 23581.156,E2 23581.156} C_VEL
LIN {X 0,Y 399.198,Z 1043.596,A -85,B 0,C 180,E1 23590.738,E2 23590.738} C_VEL
LIN {X 0,Y 401.949,Z 1066.322,A -85,B 0,C 180,E1 23599.065,E2 23599.065} C_VEL
LIN {X 0,Y 362.871,Z 1133.017,A -85,B 0,C 180,E1 23604.828,E2 23604.828} C_VEL
LIN {X 0,Y 321.55,Z 1188.172,A -85,B 0,C 180,E1 23613.225,E2 23613.225} C_VEL
LIN {X 0,Y 283.908,Z 1232.427,A -85,B 0,C 180,E1 23625.685,E2 23625.685} C_VEL
LIN {X 0,Y 260.091,Z 1261.751,A -85,B 0,C 180,E1 23641.35,E2 23641.35} C_VEL
LIN {X 0,Y 251.79,Z 1276.831,A -85,B 0,C 180,E1 23657.819,E2 23657.819} C_VEL
LIN {X 0,Y 251.117,Z 1280.091,A -85,B 0,C 180,E1 23671.733,E2 23671.733} C_VEL
LIN {X 0,Y 252.522,Z 1274.673,A -85,B 0,C 180,E1 23685.697,E2 23685.697} C_VEL
LIN {X 0,Y 264.975,Z 1255.46,A -85,B 0,C 180,E1 23702.977,E2 23702.977} C_VEL
LIN {X 0,Y 294.33,Z 1220.686,A -85,B 0,C 180,E1 23718.409,E2 23718.409} C_VEL
LIN {X 0,Y 332.998,Z 1174.045,A -85,B 0,C 180,E1 23729.433,E2 23729.433} C_VEL
LIN {X 0,Y 374.685,Z 1115.036,A -85,B 0,C 180,E1 23737.064,E2 23737.064} C_VEL
LIN {X 0,Y 402.235,Z 1066.226,A -85,B 0,C 180,E1 23740.926,E2 23740.926} C_VEL
LIN {X 0,Y 399.246,Z 1043.219,A -85,B 0,C 180,E1 23749.537,E2 23749.537} C_VEL
LIN {X 0,Y 397.632,Z 1032.224,A -85,B 0,C 180,E1 23758.844,E2 23758.844} C_VEL
LIN {X 0,Y 397.061,Z 1037.497,A -85,B 0,C 180,E1 23767.622,E2 23767.622} C_VEL
LIN {X 0,Y 398.295,Z 1055.629,A -85,B 0,C 180,E1 23776.535,E2 23776.535} C_VEL
LIN {X 0,Y 398.468,Z 1066.047,A -85,B 0,C 180,E1 23779.867,E2 23779.867} C_VEL
LIN {X 0,Y 393.365,Z 1074.925,A -85,B 0,C 180,E1 23780.409,E2 23780.409} C_VEL
LIN {X 0,Y 385.489,Z 1085.691,A -85,B 0,C 180,E1 23780.547,E2 23780.547} C_VEL
LIN {X 0,Y 344.12,Z 1146.457,A -85,B 0,C 180,E1 23787.22,E2 23787.22} C_VEL
LIN {X 0,Y 302.035,Z 1195.89,A -85,B 0,C 180,E1 23797.072,E2 23797.072} C_VEL
LIN {X 0,Y 266.8,Z 1232.95,A -85,B 0,C 180,E1 23811.25,E2 23811.25} C_VEL
LIN {X 0,Y 247.933,Z 1255.048,A -85,B 0,C 180,E1 23828.444,E2 23828.444} C_VEL
LIN {X 0,Y 243.221,Z 1263.464,A -85,B 0,C 180,E1 23844.627,E2 23844.627} C_VEL
LIN {X 0,Y 243.252,Z 1263.431,A -85,B 0,C 180,E1 23855.37,E2 23855.37} C_VEL
LIN {X 0,Y 247.877,Z 1254.956,A -85,B 0,C 180,E1 23871.558,E2 23871.558} C_VEL
LIN {X 0,Y 266.942,Z 1232.767,A -85,B 0,C 180,E1 23888.723,E2 23888.723} C_VEL
LIN {X 0,Y 302.554,Z 1195.238,A -85,B 0,C 180,E1 23902.988,E2 23902.988} C_VEL
LIN {X 0,Y 345.341,Z 1144.654,A -85,B 0,C 180,E1 23912.951,E2 23912.951} C_VEL
LIN {X 0,Y 386.011,Z 1084.7,A -85,B 0,C 180,E1 23919.387,E2 23919.387} C_VEL
LIN {X 0,Y 393.372,Z 1071.157,A -85,B 0,C 180,E1 23920.577,E2 23920.577} C_VEL
LIN {X 0,Y 393.233,Z 1049.411,A -85,B 0,C 180,E1 23929.055,E2 23929.055} C_VEL
LIN {X 0,Y 392.926,Z 1040.205,A -85,B 0,C 180,E1 23936.743,E2 23936.743} C_VEL
LIN {X 0,Y 393.613,Z 1038.991,A -85,B 0,C 180,E1 23941.168,E2 23941.168} C_VEL
LIN {X 0,Y 395.098,Z 1050.409,A -85,B 0,C 180,E1 23950.575,E2 23950.575} C_VEL
LIN {X 0,Y 396.933,Z 1071.223,A -85,B 0,C 180,E1 23958.353,E2 23958.353} C_VEL
LIN {X 0,Y 357.247,Z 1136.021,A -85,B 0,C 180,E1 23963.988,E2 23963.988} C_VEL
LIN {X 0,Y 313.717,Z 1191.838,A -85,B 0,C 180,E1 23972.778,E2 23972.778} C_VEL
LIN {X 0,Y 275.398,Z 1234.945,A -85,B 0,C 180,E1 23985.613,E2 23985.613} C_VEL
LIN {X 0,Y 251.482,Z 1263.359,A -85,B 0,C 180,E1 24001.918,E2 24001.918} C_VEL
LIN {X 0,Y 243.845,Z 1276.563,A -85,B 0,C 180,E1 24017.415,E2 24017.415} C_VEL
LIN {X 0,Y 243.129,Z 1279.829,A -85,B 0,C 180,E1 24031.79,E2 24031.79} C_VEL
LIN {X 0,Y 244.675,Z 1274.406,A -85,B 0,C 180,E1 24046.214,E2 24046.214} C_VEL
LIN {X 0,Y 258.001,Z 1255.186,A -85,B 0,C 180,E1 24063.987,E2 24063.987} C_VEL
LIN {X 0,Y 288.77,Z 1220.409,A -85,B 0,C 180,E1 24079.668,E2 24079.668} C_VEL
LIN {X 0,Y 328.936,Z 1173.593,A -85,B 0,C 180,E1 24090.727,E2 24090.727} C_VEL
LIN {X 0,Y 370.953,Z 1115.699,A -85,B 0,C 180,E1 24098.15,E2 24098.15} C_VEL
LIN {X 0,Y 397.343,Z 1069.957,A -85,B 0,C 180,E1 24101.905,E2 24101.905} C_VEL
LIN {X 0,Y 395.091,Z 1049.469,A -85,B 0,C 180,E1 24109.985,E2 24109.985} C_VEL
LIN {X 0,Y 393.743,Z 1039.251,A -85,B 0,C 180,E1 24118.833,E2 24118.833} C_VEL
LIN {X 0,Y 393.099,Z 1044.697,A -85,B 0,C 180,E1 24127.699,E2 24127.699} C_VEL
LIN {X 0,Y 393.797,Z 1063.241,A -85,B 0,C 180,E1 24136.729,E2 24136.729} C_VEL
LIN {X 0,Y 392.264,Z 1074.097,A -85,B 0,C 180,E1 24139.682,E2 24139.682} C_VEL
LIN {X 0,Y 385.489,Z 1085.691,A -85,B 0,C 180,E1 24140.547,E2 24140.547} C_VEL
LIN {X 0,Y 365.104,Z 1113.373,A -85,B 0,C 180,E1 24141.893,E2 24141.893} C_VEL
LIN {X 0,Y 321.751,Z 1169.277,A -85,B 0,C 180,E1 24149.699,E2 24149.699} C_VEL
LIN {X 0,Y 281.398,Z 1212.53,A -85,B 0,C 180,E1 24160.948,E2 24160.948} C_VEL
LIN {X 0,Y 250.384,Z 1243.841,A -85,B 0,C 180,E1 24176.927,E2 24176.927} C_VEL
LIN {X 0,Y 237.366,Z 1259.261,A -85,B 0,C 180,E1 24193.272,E2 24193.272} C_VEL
LIN {X 0,Y 235.081,Z 1264.145,A -85,B 0,C 180,E1 24208.149,E2 24208.149} C_VEL
LIN {X 0,Y 236.239,Z 1261.176,A -85,B 0,C 180,E1 24222.997,E2 24222.997} C_VEL
LIN {X 0,Y 248.305,Z 1245.932,A -85,B 0,C 180,E1 24241.31,E2 24241.31} C_VEL
LIN {X 0,Y 277.633,Z 1216.137,A -85,B 0,C 180,E1 24257.576,E2 24257.576} C_VEL
LIN {X 0,Y 319.016,Z 1172.235,A -85,B 0,C 180,E1 24269.6,E2 24269.6} C_VEL
LIN {X 0,Y 361.973,Z 1117.566,A -85,B 0,C 180,E1 24277.552,E2 24277.552} C_VEL
LIN {X 0,Y 388.495,Z 1075.584,A -85,B 0,C 180,E1 24281.363,E2 24281.363} C_VEL
LIN {X 0,Y 388.882,Z 1055.761,A -85,B 0,C 180,E1 24289.386,E2 24289.386} C_VEL
LIN {X 0,Y 389.684,Z 1045.525,A -85,B 0,C 180,E1 24298.949,E2 24298.949} C_VEL
LIN {X 0,Y 390.285,Z 1052.862,A -85,B 0,C 180,E1 24307.884,E2 24307.884} C_VEL
LIN {X 0,Y 392.078,Z 1071.543,A -85,B 0,C 180,E1 24316.359,E2 24316.359} C_VEL
LIN {X 0,Y 390.404,Z 1078.093,A -85,B 0,C 180,E1 24317.695,E2 24317.695} C_VEL
LIN {X 0,Y 349.548,Z 1141.589,A -85,B 0,C 180,E1 24323.442,E2 24323.442} C_VEL
LIN {X 0,Y 305.584,Z 1195.62,A -85,B 0,C 180,E1 24332.378,E2 24332.378} C_VEL
LIN {X 0,Y 267.282,Z 1236.896,A -85,B 0,C 180,E1 24345.331,E2 24345.331} C_VEL
LIN {X 0,Y 242.511,Z 1265.285,A -85,B 0,C 180,E1 24363.01,E2 24363.01} C_VEL
LIN {X 0,Y 235.282,Z 1277.981,A -85,B 0,C 180,E1 24380.718,E2 24380.718} C_VEL
LIN {X 0,Y 235.125,Z 1279.566,A -85,B 0,C 180,E1 24391.851,E2 24391.851} C_VEL
LIN {X 0,Y 236.816,Z 1274.137,A -85,B 0,C 180,E1 24406.768,E2 24406.768} C_VEL
LIN {X 0,Y 251.363,Z 1254.595,A -85,B 0,C 180,E1 24425.257,E2 24425.257} C_VEL
LIN {X 0,Y 283.328,Z 1220.131,A -85,B 0,C 180,E1 24440.982,E2 24440.982} C_VEL
LIN {X 0,Y 326.055,Z 1171.933,A -85,B 0,C 180,E1 24452.248,E2 24452.248} C_VEL
LIN {X 0,Y 369.944,Z 1112.295,A -85,B 0,C 180,E1 24459.65,E2 24459.65} C_VEL
LIN {X 0,Y 392.385,Z 1074.731,A -85,B 0,C 180,E1 24462.582,E2 24462.582} C_VEL
LIN {X 0,Y 390.655,Z 1054.722,A -85,B 0,C 180,E1 24470.998,E2 24470.998} C_VEL
LIN {X 0,Y 389.828,Z 1046.302,A -85,B 0,C 180,E1 24478.821,E2 24478.821} C_VEL
LIN {X 0,Y 389.016,Z 1050.406,A -85,B 0,C 180,E1 24486.653,E2 24486.653} C_VEL
LIN {X 0,Y 389.048,Z 1066.874,A -85,B 0,C 180,E1 24495.511,E2 24495.511} C_VEL
LIN {X 0,Y 387.758,Z 1077.627,A -85,B 0,C 180,E1 24498.785,E2 24498.785} C_VEL
LIN {X 0,Y 365.104,Z 1113.373,A -85,B 0,C 180,E1 24501.893,E2 24501.893} C_VEL
LIN {X 0,Y 343.202,Z 1139.162,A -85,B 0,C 180,E1 24503.635,E2 24503.635} C_VEL
LIN {X 0,Y 298.293,Z 1190.439,A -85,B 0,C 180,E1 24512.885,E2 24512.885} C_VEL
LIN {X 0,Y 258.946,Z 1228.986,A -85,B 0,C 180,E1 24526.458,E2 24526.458} C_VEL
LIN {X 0,Y 235.471,Z 1252.329,A -85,B 0,C 180,E1 24543.172,E2 24543.172} C_VEL
LIN {X 0,Y 227.534,Z 1263.015,A -85,B 0,C 180,E1 24560.397,E2 24560.397} C_VEL
LIN {X 0,Y 227.246,Z 1263.959,A -85,B 0,C 180,E1 24575.75,E2 24575.75} C_VEL
LIN {X 0,Y 232.716,Z 1255.495,A -85,B 0,C 180,E1 24593.041,E2 24593.041} C_VEL
LIN {X 0,Y 254.22,Z 1233.314,A -85,B 0,C 180,E1 24611.061,E2 24611.061} C_VEL
LIN {X 0,Y 292.519,Z 1196.133,A -85,B 0,C 180,E1 24625.488,E2 24625.488} C_VEL
LIN {X 0,Y 337.195,Z 1146.385,A -85,B 0,C 180,E1 24635.27,E2 24635.27} C_VEL
LIN {X 0,Y 379.694,Z 1086.661,A -85,B 0,C 180,E1 24641.573,E2 24641.573} C_VEL
LIN {X 0,Y 383.703,Z 1079.841,A -85,B 0,C 180,E1 24642.224,E2 24642.224} C_VEL
LIN {X 0,Y 384.549,Z 1061.907,A -85,B 0,C 180,E1 24649.839,E2 24649.839} C_VEL
LIN {X 0,Y 385.629,Z 1052.508,A -85,B 0,C 180,E1 24658.938,E2 24658.938} C_VEL
LIN {X 0,Y 385.996,Z 1059.889,A -85,B 0,C 180,E1 24667.973,E2 24667.973} C_VEL
LIN {X 0,Y 387.113,Z 1078.893,A -85,B 0,C 180,E1 24676.49,E2 24676.49} C_VEL
LIN {X 0,Y 344.023,Z 1144.352,A -85,B 0,C 180,E1 24682.543,E2 24682.543} C_VEL
LIN {X 0,Y 298.703,Z 1198.051,A -85,B 0,C 180,E1 24691.649,E2 24691.649} C_VEL
LIN {X 0,Y 259.522,Z 1238.511,A -85,B 0,C 180,E1 24704.884,E2 24704.884} C_VEL
LIN {X 0,Y 234.393,Z 1266.014,A -85,B 0,C 180,E1 24723.041,E2 24723.041} C_VEL
LIN {X 0,Y 227.297,Z 1277.715,A -85,B 0,C 180,E1 24740.389,E2 24740.389} C_VEL
LIN {X 0,Y 227.115,Z 1279.303,A -85,B 0,C 180,E1 24751.916,E2 24751.916} C_VEL
LIN {X 0,Y 228.982,Z 1273.868,A -85,B 0,C 180,E1 24767.359,E2 24767.359} C_VEL
LIN {X 0,Y 244.271,Z 1254.638,A -85,B 0,C 180,E1 24786.188,E2 24786.188} C_VEL
LIN {X 0,Y 278.054,Z 1219.854,A -85,B 0,C 180,E1 24802.343,E2 24802.343} C_VEL
LIN {X 0,Y 321.38,Z 1172.696,A -85,B 0,C 180,E1 24813.392,E2 24813.392} C_VEL
LIN {X 0,Y 365.673,Z 1114.248,A -85,B 0,C 180,E1 24820.664,E2 24820.664} C_VEL
LIN {X 0,Y 387.41,Z 1078.854,A -85,B 0,C 180,E1 24823.484,E2 24823.484} C_VEL
LIN {X 0,Y 386.162,Z 1060.013,A -85,B 0,C 180,E1 24832.031,E2 24832.031} C_VEL
LIN {X 0,Y 385.685,Z 1052.888,A -85,B 0,C 180,E1 24841.062,E2 24841.062} C_VEL
LIN {X 0,Y 384.61,Z 1063.372,A -85,B 0,C 180,E1 24850.734,E2 24850.734} C_VEL
LIN {X 0,Y 383.877,Z 1079.537,A -85,B 0,C 180,E1 24857.553,E2 24857.553} C_VEL
LIN {X 0,Y 343.202,Z 1139.162,A -85,B 0,C 180,E1 24863.635,E2 24863.635} C_VEL
LIN {X 0,Y 320.084,Z 1162.887,A -85,B 0,C 180,E1 24865.853,E2 24865.853} C_VEL
LIN {X 0,Y 275.046,Z 1208.94,A -85,B 0,C 180,E1 24876.837,E2 24876.837} C_VEL
LIN {X 0,Y 239.129,Z 1241.959,A -85,B 0,C 180,E1 24892.906,E2 24892.906} C_VEL
LIN {X 0,Y 221.812,Z 1259.795,A -85,B 0,C 180,E1 24912.061,E2 24912.061} C_VEL
LIN {X 0,Y 219.095,Z 1264.67,A -85,B 0,C 180,E1 24928.013,E2 24928.013} C_VEL
LIN {X 0,Y 220.47,Z 1261.709,A -85,B 0,C 180,E1 24943.945,E2 24943.945} C_VEL
LIN {X 0,Y 234.264,Z 1246.479,A -85,B 0,C 180,E1 24963.423,E2 24963.423} C_VEL
LIN {X 0,Y 266.643,Z 1216.689,A -85,B 0,C 180,E1 24980.228,E2 24980.228} C_VEL
LIN {X 0,Y 310.975,Z 1172.784,A -85,B 0,C 180,E1 24992.227,E2 24992.227} C_VEL
LIN {X 0,Y 356.52,Z 1117.405,A -85,B 0,C 180,E1 25000.082,E2 25000.082} C_VEL
LIN {X 0,Y 378.832,Z 1083.746,A -85,B 0,C 180,E1 25003.205,E2 25003.205} C_VEL
LIN {X 0,Y 380.355,Z 1065.366,A -85,B 0,C 180,E1 25012.041,E2 25012.041} C_VEL
LIN {X 0,Y 381.405,Z 1059.363,A -85,B 0,C 180,E1 25018.927,E2 25018.927} C_VEL
LIN {X 0,Y 381.693,Z 1066.938,A -85,B 0,C 180,E1 25028.063,E2 25028.063} C_VEL
LIN {X 0,Y 382.252,Z 1083.395,A -85,B 0,C 180,E1 25035.706,E2 25035.706} C_VEL
LIN {X 0,Y 339.231,Z 1146.261,A -85,B 0,C 180,E1 25041.509,E2 25041.509} C_VEL
LIN {X 0,Y 292.943,Z 1199.297,A -85,B 0,C 180,E1 25050.602,E2 25050.602} C_VEL
LIN {X 0,Y 251.332,Z 1240.578,A -85,B 0,C 180,E1 25064.618,E2 25064.618} C_VEL
LIN {X 0,Y 226.961,Z 1265.739,A -85,B 0,C 180,E1 25082.082,E2 25082.082} C_VEL
LIN {X 0,Y 219.321,Z 1277.449,A -85,B 0,C 180,E1 25100.036,E2 25100.036} C_VEL
LIN {X 0,Y 219.108,Z 1279.04,A -85,B 0,C 180,E1 25111.986,E2 25111.986} C_VEL
LIN {X 0,Y 221.161,Z 1273.599,A -85,B 0,C 180,E1 25127.994,E2 25127.994} C_VEL
LIN {X 0,Y 237.501,Z 1254.362,A -85,B 0,C 180,E1 25147.392,E2 25147.392} C_VEL
LIN {X 0,Y 272.958,Z 1219.578,A -85,B 0,C 180,E1 25163.752,E2 25163.752} C_VEL
LIN {X 0,Y 318.397,Z 1171.633,A -85,B 0,C 180,E1 25174.872,E2 25174.872} C_VEL
LIN {X 0,Y 364.064,Z 1112.407,A -85,B 0,C 180,E1 25182.041,E2 25182.041} C_VEL
LIN {X 0,Y 382.523,Z 1082.874,A -85,B 0,C 180,E1 25184.452,E2 25184.452} C_VEL
LIN {X 0,Y 381.754,Z 1065.376,A -85,B 0,C 180,E1 25193.087,E2 25193.087} C_VEL
LIN {X 0,Y 381.463,Z 1059.741,A -85,B 0,C 180,E1 25201.074,E2 25201.074} C_VEL
LIN {X 0,Y 380.063,Z 1069.391,A -85,B 0,C 180,E1 25210.282,E2 25210.282} C_VEL
LIN {X 0,Y 378.661,Z 1084.855,A -85,B 0,C 180,E1 25216.96,E2 25216.96} C_VEL
LIN {X 0,Y 336.049,Z 1144.237,A -85,B 0,C 180,E1 25223.006,E2 25223.006} C_VEL
LIN {X 0,Y 320.084,Z 1162.887,A -85,B 0,C 180,E1 25225.853,E2 25225.853} C_VEL
LIN {X 0,Y 296.111,Z 1184.476,A -85,B 0,C 180,E1 25228.615,E2 25228.615} C_VEL
LIN {X 0,Y 252.994,Z 1224.429,A -85,B 0,C 180,E1 25241.401,E2 25241.401} C_VEL
LIN {X 0,Y 222.818,Z 1251.007,A -85,B 0,C 180,E1 25259.269,E2 25259.269} C_VEL
LIN {X 0,Y 212.502,Z 1262.03,A -85,B 0,C 180,E1 25275.519,E2 25275.519} C_VEL
LIN {X 0,Y 211.299,Z 1264.916,A -85,B 0,C 180,E1 25292.057,E2 25292.057} C_VEL
LIN {X 0,Y 215.163,Z 1258.831,A -85,B 0,C 180,E1 25310.656,E2 25310.656} C_VEL
LIN {X 0,Y 234.165,Z 1240.554,A -85,B 0,C 180,E1 25329.417,E2 25329.417} C_VEL
LIN {X 0,Y 272.506,Z 1206.859,A -85,B 0,C 180,E1 25345.255,E2 25345.255} C_VEL
LIN {X 0,Y 319.83,Z 1159.339,A -85,B 0,C 180,E1 25356.024,E2 25356.024} C_VEL
LIN {X 0,Y 364.554,Z 1102.673,A -85,B 0,C 180,E1 25362.715,E2 25362.715} C_VEL
LIN {X 0,Y 374.038,Z 1087.554,A -85,B 0,C 180,E1 25364.265,E2 25364.265} C_VEL
LIN {X 0,Y 375.971,Z 1070.68,A -85,B 0,C 180,E1 25373.114,E2 25373.114} C_VEL
LIN {X 0,Y 377.208,Z 1066.709,A -85,B 0,C 180,E1 25381.219,E2 25381.219} C_VEL
LIN {X 0,Y 377.302,Z 1077.807,A -85,B 0,C 180,E1 25390.492,E2 25390.492} C_VEL
LIN {X 0,Y 376.251,Z 1089.662,A -85,B 0,C 180,E1 25395.013,E2 25395.013} C_VEL
LIN {X 0,Y 331.008,Z 1152.425,A -85,B 0,C 180,E1 25400.986,E2 25400.986} C_VEL
LIN {X 0,Y 284.488,Z 1203.31,A -85,B 0,C 180,E1 25410.222,E2 25410.222} C_VEL
LIN {X 0,Y 243.423,Z 1242.157,A -85,B 0,C 180,E1 25424.177,E2 25424.177} C_VEL
LIN {X 0,Y 218.062,Z 1267.372,A -85,B 0,C 180,E1 25443.096,E2 25443.096} C_VEL
LIN {X 0,Y 211.348,Z 1277.183,A -85,B 0,C 180,E1 25459.656,E2 25459.656} C_VEL
LIN {X 0,Y 211.097,Z 1278.777,A -85,B 0,C 180,E1 25472.062,E2 25472.062} C_VEL
LIN {X 0,Y 213.378,Z 1273.331,A -85,B 0,C 180,E1 25488.674,E2 25488.674} C_VEL
LIN {X 0,Y 230.847,Z 1254.085,A -85,B 0,C 180,E1 25508.665,E2 25508.665} C_VEL
LIN {X 0,Y 268.035,Z 1219.301,A -85,B 0,C 180,E1 25525.213,E2 25525.213} C_VEL
LIN {X 0,Y 314.501,Z 1171.856,A -85,B 0,C 180,E1 25536.169,E2 25536.169} C_VEL
LIN {X 0,Y 361.578,Z 1112.137,A -85,B 0,C 180,E1 25543.299,E2 25543.299} C_VEL
LIN {X 0,Y 377.62,Z 1087.643,A -85,B 0,C 180,E1 25545.21,E2 25545.21} C_VEL
LIN {X 0,Y 377.288,Z 1070.799,A -85,B 0,C 180,E1 25554.164,E2 25554.164} C_VEL
LIN {X 0,Y 377.247,Z 1066.583,A -85,B 0,C 180,E1 25561.086,E2 25561.086} C_VEL
LIN {X 0,Y 375.407,Z 1076.346,A -85,B 0,C 180,E1 25570.411,E2 25570.411} C_VEL
LIN {X 0,Y 373.311,Z 1089.82,A -85,B 0,C 180,E1 25576.117,E2 25576.117} C_VEL
LIN {X 0,Y 328.45,Z 1149.706,A -85,B 0,C 180,E1 25582.418,E2 25582.418} C_VEL
LIN {X 0,Y 296.111,Z 1184.476,A -85,B 0,C 180,E1 25588.615,E2 25588.615} C_VEL
LIN {X 0,Y 271.811,Z 1203.795,A -85,B 0,C 180,E1 25592.097,E2 25592.097} C_VEL
LIN {X 0,Y 230.639,Z 1238.609,A -85,B 0,C 180,E1 25607.571,E2 25607.571} C_VEL
LIN {X 0,Y 208.812,Z 1257.899,A -85,B 0,C 180,E1 25626.429,E2 25626.429} C_VEL
LIN {X 0,Y 203.244,Z 1264.782,A -85,B 0,C 180,E1 25643.566,E2 25643.566} C_VEL
LIN {X 0,Y 203.282,Z 1264.751,A -85,B 0,C 180,E1 25656.431,E2 25656.431} C_VEL
LIN {X 0,Y 210.526,Z 1256.064,A -85,B 0,C 180,E1 25676.004,E2 25676.004} C_VEL
LIN {X 0,Y 238.522,Z 1232.187,A -85,B 0,C 180,E1 25696.118,E2 25696.118} C_VEL
LIN {X 0,Y 281.718,Z 1194.619,A -85,B 0,C 180,E1 25710.334,E2 25710.334} C_VEL
LIN {X 0,Y 330.072,Z 1144.428,A -85,B 0,C 180,E1 25719.571,E2 25719.571} C_VEL
LIN {X 0,Y 369.206,Z 1092.131,A -85,B 0,C 180,E1 25725.077,E2 25725.077} C_VEL
LIN {X 0,Y 371.364,Z 1077.499,A -85,B 0,C 180,E1 25733.028,E2 25733.028} C_VEL
LIN {X 0,Y 372.712,Z 1073.383,A -85,B 0,C 180,E1 25741.233,E2 25741.233} C_VEL
LIN {X 0,Y 372.615,Z 1084.813,A -85,B 0,C 180,E1 25750.626,E2 25750.626} C_VEL
LIN {X 0,Y 371.239,Z 1093.93,A -85,B 0,C 180,E1 25754.11,E2 25754.11} C_VEL
LIN {X 0,Y 324.255,Z 1156.619,A -85,B 0,C 180,E1 25760.212,E2 25760.212} C_VEL
LIN {X 0,Y 275.495,Z 1207.616,A -85,B 0,C 180,E1 25769.934,E2 25769.934} C_VEL
LIN {X 0,Y 234.006,Z 1245.042,A -85,B 0,C 180,E1 25784.471,E2 25784.471} C_VEL
LIN {X 0,Y 209.175,Z 1268.739,A -85,B 0,C 180,E1 25804.189,E2 25804.189} C_VEL
LIN {X 0,Y 203.087,Z 1278.016,A -85,B 0,C 180,E1 25823.563,E2 25823.563} C_VEL
LIN {X 0,Y 203.035,Z 1278.022,A -85,B 0,C 180,E1 25836.441,E2 25836.441} C_VEL
LIN {X 0,Y 208.877,Z 1268.921,A -85,B 0,C 180,E1 25855.624,E2 25855.624} C_VEL
LIN {X 0,Y 233.898,Z 1245.096,A -85,B 0,C 180,E1 25875.559,E2 25875.559} C_VEL
LIN {X 0,Y 276.537,Z 1206.684,A -85,B 0,C 180,E1 25890.356,E2 25890.356} C_VEL
LIN {X 0,Y 325.792,Z 1155.078,A -85,B 0,C 180,E1 25899.991,E2 25899.991} C_VEL
LIN {X 0,Y 372.562,Z 1091.918,A -85,B 0,C 180,E1 25906.151,E2 25906.151} C_VEL
LIN {X 0,Y 372.716,Z 1077.554,A -85,B 0,C 180,E1 25914.092,E2 25914.092} C_VEL
LIN {X 0,Y 372.731,Z 1073.255,A -85,B 0,C 180,E1 25921.099,E2 25921.099} C_VEL
LIN {X 0,Y 370.641,Z 1083.308,A -85,B 0,C 180,E1 25930.546,E2 25930.546} C_VEL
LIN {X 0,Y 368.014,Z 1094.848,A -85,B 0,C 180,E1 25935.261,E2 25935.261} C_VEL
LIN {X 0,Y 322.405,Z 1153.438,A -85,B 0,C 180,E1 25941.567,E2 25941.567} C_VEL
LIN {X 0,Y 275.141,Z 1200.778,A -85,B 0,C 180,E1 25951.213,E2 25951.213} C_VEL
LIN {X 0,Y 271.811,Z 1203.795,A -85,B 0,C 180,E1 25952.097,E2 25952.097} C_VEL
